C05478=1167.973,405.826,-85.740,-176.090,9.388,148.780
C05479=1167.977,405.579,-85.703,-176.089,9.386,148.779
C05480=1167.980,405.332,-85.667,-176.089,9.384,148.778
C05481=1167.985,405.085,-85.630,-176.088,9.382,148.778
C05482=1167.988,404.838,-85.594,-176.088,9.380,148.777
C05483=1167.992,404.590,-85.558,-176.088,9.378,148.776
C05484=1167.996,404.343,-85.522,-176.087,9.376,148.776
C05485=1168.000,404.095,-85.486,-176.087,9.373,148.775
C05486=1168.003,403.848,-85.449,-176.086,9.372,148.774
C05487=1168.008,403.600,-85.413,-176.086,9.369,148.774
C05488=1168.011,403.354,-85.377,-176.086,9.368,148.773
C05489=1168.016,403.106,-85.341,-176.086,9.365,148.773
C05490=1168.019,402.859,-85.304,-176.085,9.363,148.772
C05491=1168.023,402.611,-85.268,-176.085,9.361,148.771
C05492=1168.027,402.364,-85.231,-176.084,9.359,148.771
C05493=1168.031,402.116,-85.196,-176.084,9.357,148.770
C05494=1168.035,401.869,-85.159,-176.083,9.355,148.769
C05495=1168.039,401.622,-85.124,-176.083,9.352,148.768
C05496=1168.043,401.375,-85.087,-176.082,9.350,148.768
C05497=1168.047,401.127,-85.051,-176.082,9.348,148.767
C05498=1168.051,400.880,-85.014,-176.081,9.346,148.766
C05499=1168.054,400.632,-84.979,-176.081,9.344,148.766
C05500=1168.058,400.385,-84.942,-176.081,9.341,148.765
C05501=1168.062,400.138,-84.906,-176.080,9.339,148.764
C05502=1168.067,399.891,-84.870,-176.080,9.337,148.764
C05503=1168.070,399.644,-84.834,-176.080,9.334,148.763
C05504=1168.075,399.396,-84.797,-176.079,9.332,148.762
C05505=1168.078,399.149,-84.762,-176.079,9.330,148.762
C05506=1168.082,398.902,-84.725,-176.079,9.327,148.761
C05507=1168.086,398.654,-84.689,-176.078,9.326,148.760
C05508=1168.090,398.407,-84.653,-176.078,9.323,148.759
C05509=1168.094,398.160,-84.617,-176.078,9.320,148.759
C05510=1168.098,397.912,-84.580,-176.078,9.317,148.758
C05511=1168.101,397.665,-84.545,-176.077,9.316,148.757
C05512=1168.106,397.417,-84.508,-176.077,9.313,148.757
C05513=1168.109,397.170,-84.472,-176.077,9.311,148.756
C05514=1168.113,396.923,-84.437,-176.076,9.308,148.755
C05515=1168.117,396.676,-84.400,-176.076,9.305,148.754
C05516=1168.121,396.428,-84.364,-176.075,9.304,148.754
C05517=1168.125,396.181,-84.327,-176.075,9.301,148.753
C05518=1168.128,395.933,-84.292,-176.075,9.298,148.752
C05519=1168.133,395.686,-84.255,-176.075,9.296,148.751
C05520=1168.136,395.439,-84.219,-176.074,9.293,148.751
C05521=1168.141,395.191,-84.183,-176.074,9.291,148.750
C05522=1168.144,394.944,-84.147,-176.074,9.288,148.749
C05523=1168.148,394.696,-84.111,-176.074,9.285,148.749
C05524=1168.152,394.449,-84.075,-176.074,9.283,148.748
C05525=1168.156,394.201,-84.038,-176.073,9.280,148.747
C05526=1168.160,393.955,-84.003,-176.073,9.277,148.746
C05527=1168.164,393.708,-83.967,-176.073,9.275,148.746
C05528=1168.168,393.460,-83.931,-176.073,9.272,148.745
C05529=1168.171,393.213,-83.895,-176.073,9.270,148.744
C05530=1168.176,392.965,-83.859,-176.073,9.267,148.743
C05531=1168.180,392.718,-83.823,-176.072,9.265,148.743
C05532=1168.184,392.471,-83.786,-176.073,9.261,148.742
C05533=1168.187,392.223,-83.751,-176.072,9.258,148.741
C05534=1168.191,391.938,-83.708,-176.072,9.256,148.740
C05535=1168.196,391.653,-83.667,-176.072,9.252,148.739
C05536=1168.201,391.368,-83.626,-176.073,9.249,148.739
C05537=1168.205,391.083,-83.584,-176.072,9.246,148.738
C05538=1168.209,390.835,-83.549,-176.072,9.242,148.737
C05539=1168.213,390.588,-83.512,-176.072,9.240,148.736
C05540=1168.216,390.341,-83.476,-176.072,9.237,148.735
C05541=1168.221,390.093,-83.441,-176.073,9.234,148.735
C05542=1168.225,389.847,-83.404,-176.072,9.231,148.734
C05543=1168.228,389.599,-83.369,-176.073,9.228,148.733
C05544=1168.233,389.351,-83.333,-176.073,9.225,148.732
C05545=1168.236,389.104,-83.297,-176.073,9.222,148.731
C05546=1168.241,388.857,-83.260,-176.073,9.219,148.731
C05547=1168.244,388.609,-83.225,-176.073,9.216,148.730
C05548=1168.248,388.362,-83.189,-176.073,9.213,148.729
C05549=1168.252,388.114,-83.152,-176.073,9.210,148.729
C05550=1168.256,387.867,-83.117,-176.073,9.207,148.728
C05551=1168.259,387.619,-83.081,-176.074,9.204,148.727
C05552=1168.264,387.372,-83.045,-176.074,9.201,148.726
C05553=1168.268,387.125,-83.009,-176.075,9.197,148.726
C05554=1168.271,386.878,-82.974,-176.075,9.195,148.725
C05555=1168.276,386.630,-82.937,-176.075,9.191,148.724
C05556=1168.279,386.383,-82.902,-176.075,9.188,148.723
C05557=1168.283,386.136,-82.866,-176.076,9.185,148.723
C05558=1168.287,385.888,-82.829,-176.076,9.181,148.722
C05559=1168.291,385.640,-82.794,-176.077,9.178,148.721
C05560=1168.294,385.393,-82.758,-176.077,9.176,148.721
C05561=1168.299,385.146,-82.723,-176.077,9.172,148.720
C05562=1168.303,384.899,-82.686,-176.078,9.169,148.719
C05563=1168.306,384.651,-82.651,-176.078,9.165,148.718
C05564=1168.311,384.404,-82.615,-176.080,9.161,148.718
C05565=1168.315,384.156,-82.579,-176.080,9.158,148.717
C05566=1168.318,383.909,-82.544,-176.081,9.155,148.716
C05567=1168.322,383.661,-82.508,-176.081,9.152,148.716
C05568=1168.327,383.415,-82.471,-176.082,9.148,148.715
C05569=1168.330,383.167,-82.436,-176.083,9.145,148.714
C05570=1168.334,382.920,-82.400,-176.083,9.142,148.713
C05571=1168.338,382.672,-82.364,-176.084,9.138,148.713
C05572=1168.342,382.424,-82.329,-176.085,9.134,148.712
C05573=1168.346,382.177,-82.293,-176.085,9.131,148.711
C05574=1168.349,381.929,-82.258,-176.086,9.128,148.711
C05575=1168.354,381.682,-82.222,-176.087,9.124,148.710
C05576=1168.358,381.435,-82.186,-176.088,9.121,148.709
C05577=1168.362,381.187,-82.151,-176.089,9.118,148.709
C05578=1168.365,380.940,-82.115,-176.090,9.113,148.708
C05579=1168.370,380.692,-82.079,-176.091,9.110,148.707
C05580=1168.374,380.445,-82.044,-176.092,9.106,148.707
C05581=1168.377,380.198,-82.008,-176.093,9.103,148.706
C05582=1168.381,379.951,-81.972,-176.093,9.100,148.705
C05583=1168.385,379.703,-81.937,-176.095,9.096,148.705
C05584=1168.389,379.455,-81.900,-176.095,9.093,148.704
C05585=1168.394,379.208,-81.866,-176.097,9.089,148.703
C05586=1168.397,378.960,-81.830,-176.098,9.085,148.703
C05587=1168.401,378.713,-81.795,-176.099,9.082,148.702
C05588=1168.405,378.465,-81.759,-176.100,9.078,148.701
C05589=1168.409,378.218,-81.723,-176.101,9.075,148.701
C05590=1168.413,377.971,-81.688,-176.103,9.071,148.700
C05591=1168.417,377.723,-81.652,-176.104,9.067,148.700
C05592=1168.421,377.476,-81.617,-176.104,9.063,148.699
C05593=1168.424,377.228,-81.581,-176.106,9.060,148.698
C05594=1168.428,376.982,-81.546,-176.108,9.056,148.698
C05595=1168.432,376.734,-81.511,-176.109,9.053,148.697
C05596=1168.436,376.487,-81.475,-176.110,9.049,148.697
C05597=1168.441,376.238,-81.440,-176.111,9.045,148.696
C05598=1168.445,375.991,-81.404,-176.113,9.041,148.695
C05599=1168.448,375.744,-81.369,-176.114,9.038,148.695
C05600=1168.452,375.496,-81.333,-176.115,9.034,148.694
C05601=1168.456,375.249,-81.298,-176.117,9.031,148.694
C05602=1168.460,375.002,-81.263,-176.118,9.027,148.693
C05603=1168.464,374.754,-81.228,-176.120,9.023,148.692
C05604=1168.468,374.506,-81.192,-176.121,9.019,148.692
C05605=1168.471,374.259,-81.157,-176.123,9.016,148.691
C05606=1168.476,374.012,-81.121,-176.124,9.012,148.691
C05607=1168.480,373.764,-81.087,-176.125,9.008,148.690
C05608=1168.483,373.516,-81.051,-176.127,9.005,148.690
C05609=1168.487,373.270,-81.016,-176.129,9.001,148.689
C05610=1168.491,373.022,-80.980,-176.130,8.997,148.689
C05611=1168.495,372.774,-80.946,-176.132,8.993,148.688
C05612=1168.499,372.527,-80.910,-176.134,8.990,148.688
C05613=1168.503,372.280,-80.875,-176.135,8.986,148.687
C05614=1168.507,372.032,-80.840,-176.137,8.982,148.687
C05615=1168.511,371.784,-80.804,-176.138,8.978,148.686
C05616=1168.515,371.537,-80.769,-176.140,8.975,148.686
C05617=1168.519,371.289,-80.734,-176.142,8.971,148.685
C05618=1168.523,371.042,-80.699,-176.144,8.967,148.684
C05619=1168.527,370.794,-80.664,-176.145,8.963,148.684
C05620=1168.531,370.547,-80.629,-176.147,8.960,148.684
C05621=1168.535,370.300,-80.594,-176.150,8.955,148.683
C05622=1168.539,370.052,-80.559,-176.151,8.951,148.683
C05623=1168.543,369.804,-80.523,-176.153,8.948,148.682
C05624=1168.547,369.557,-80.489,-176.155,8.944,148.682
C05625=1168.551,369.309,-80.453,-176.157,8.941,148.681
C05626=1168.555,369.061,-80.418,-176.159,8.937,148.681
C05627=1168.559,368.815,-80.383,-176.160,8.933,148.680
C05628=1168.562,368.567,-80.349,-176.162,8.929,148.680
C05629=1168.567,368.320,-80.314,-176.164,8.925,148.679
C05630=1168.571,368.072,-80.279,-176.166,8.922,148.679
C05631=1168.574,367.824,-80.243,-176.168,8.918,148.678
C05632=1168.579,367.577,-80.209,-176.170,8.914,148.678
C05633=1168.583,367.329,-80.173,-176.172,8.910,148.678
C05634=1168.587,367.082,-80.139,-176.174,8.907,148.677
C05635=1168.591,366.834,-80.104,-176.176,8.903,148.677
C05636=1168.594,366.587,-80.069,-176.178,8.899,148.676
C05637=1168.599,366.339,-80.035,-176.180,8.896,148.676
C05638=1168.603,366.057,-79.995,-176.182,8.891,148.676
C05639=1168.607,365.775,-79.955,-176.185,8.887,148.675
C05640=1168.612,365.493,-79.916,-176.187,8.882,148.675
C05641=1168.616,365.211,-79.876,-176.190,8.878,148.674
C05642=1168.620,364.962,-79.841,-176.192,8.874,148.674
C05643=1168.625,364.715,-79.806,-176.194,8.871,148.673
C05644=1168.628,364.468,-79.771,-176.196,8.867,148.673
C05645=1168.632,364.220,-79.737,-176.198,8.863,148.673
C05646=1168.636,363.972,-79.702,-176.200,8.860,148.672
C05647=1168.641,363.725,-79.668,-176.203,8.855,148.672
C05648=1168.644,363.478,-79.633,-176.205,8.852,148.671
C05649=1168.648,363.230,-79.598,-176.207,8.849,148.671
C05650=1168.652,362.982,-79.564,-176.209,8.844,148.671
C05651=1168.656,362.735,-79.530,-176.211,8.840,148.670
C05652=1168.660,362.487,-79.495,-176.214,8.837,148.670
C05653=1168.665,362.239,-79.460,-176.216,8.833,148.670
C05654=1168.668,361.992,-79.425,-176.218,8.829,148.669
C05655=1168.672,361.745,-79.391,-176.220,8.826,148.669
C05656=1168.676,361.497,-79.356,-176.223,8.822,148.669
C05657=1168.680,361.250,-79.322,-176.225,8.818,148.668
C05658=1168.684,361.002,-79.287,-176.227,8.815,148.668
C05659=1168.688,360.754,-79.253,-176.230,8.810,148.668
C05660=1168.692,360.506,-79.219,-176.232,8.807,148.667
C05661=1168.696,360.259,-79.184,-176.234,8.803,148.667
C05662=1168.700,360.011,-79.150,-176.237,8.799,148.667
C05663=1168.704,359.764,-79.116,-176.239,8.796,148.666
C05664=1168.709,359.516,-79.081,-176.241,8.792,148.666
C05665=1168.712,359.268,-79.047,-176.244,8.788,148.666
C05666=1168.716,359.021,-79.012,-176.245,8.785,148.665
C05667=1168.720,358.773,-78.978,-176.248,8.781,148.665
C05668=1168.724,358.526,-78.944,-176.251,8.777,148.665
C05669=1168.727,358.278,-78.909,-176.252,8.774,148.664
C05670=1168.732,358.031,-78.875,-176.255,8.770,148.664
C05671=1168.736,357.783,-78.841,-176.258,8.766,148.664
C05672=1168.740,357.535,-78.806,-176.259,8.763,148.663
C05673=1168.744,357.288,-78.772,-176.262,8.759,148.663
C05674=1168.748,357.039,-78.738,-176.265,8.755,148.663
C05675=1168.752,356.792,-78.704,-176.266,8.752,148.663
C05676=1168.756,356.545,-78.670,-176.269,8.748,148.662
C05677=1168.760,356.297,-78.636,-176.272,8.744,148.662
C05678=1168.764,356.050,-78.601,-176.274,8.741,148.662
C05679=1168.768,355.803,-78.567,-176.276,8.737,148.661
C05680=1168.772,355.554,-78.533,-176.278,8.734,148.661
C05681=1168.776,355.307,-78.499,-176.281,8.730,148.661
C05682=1168.780,355.060,-78.465,-176.283,8.727,148.661
C05683=1168.784,354.812,-78.431,-176.285,8.723,148.660
C05684=1168.788,354.564,-78.398,-176.288,8.719,148.660
C05685=1168.793,354.316,-78.363,-176.290,8.716,148.660
C05686=1168.796,354.069,-78.329,-176.292,8.712,148.660
C05687=1168.801,353.821,-78.295,-176.295,8.708,148.659
C05688=1168.805,353.573,-78.261,-176.297,8.705,148.659
C05689=1168.808,353.326,-78.227,-176.299,8.701,148.659
C05690=1168.813,353.078,-78.193,-176.302,8.698,148.658
C05691=1168.817,352.830,-78.159,-176.305,8.694,148.658
C05692=1168.820,352.583,-78.125,-176.306,8.690,148.658
C05693=1168.825,352.335,-78.091,-176.309,8.687,148.658
C05694=1168.828,352.088,-78.057,-176.312,8.683,148.657
C05695=1168.833,351.840,-78.024,-176.314,8.680,148.657
C05696=1168.837,351.592,-77.989,-176.316,8.676,148.657
C05697=1168.841,351.344,-77.956,-176.318,8.673,148.657
C05698=1168.845,351.097,-77.922,-176.321,8.669,148.656
C05699=1168.849,350.849,-77.889,-176.323,8.665,148.656
C05700=1168.853,350.601,-77.854,-176.325,8.662,148.656
C05701=1168.857,350.353,-77.821,-176.328,8.658,148.656
C05702=1168.861,350.106,-77.787,-176.331,8.655,148.655
C05703=1168.865,349.858,-77.754,-176.333,8.651,148.655
C05704=1168.869,349.610,-77.719,-176.335,8.648,148.655
C05705=1168.873,349.363,-77.686,-176.338,8.643,148.654
C05706=1168.877,349.115,-77.652,-176.340,8.640,148.654
C05707=1168.881,348.868,-77.619,-176.342,8.637,148.654
C05708=1168.886,348.620,-77.586,-176.344,8.634,148.654
C05709=1168.889,348.372,-77.551,-176.347,8.629,148.653
C05710=1168.893,348.124,-77.518,-176.350,8.626,148.653
C05711=1168.897,347.876,-77.485,-176.352,8.623,148.653
C05712=1168.901,347.629,-77.451,-176.354,8.620,148.653
C05713=1168.906,347.381,-77.417,-176.357,8.615,148.653
C05714=1168.910,347.134,-77.384,-176.359,8.612,148.652
C05715=1168.913,346.886,-77.350,-176.362,8.609,148.652
C05716=1168.917,346.638,-77.317,-176.364,8.606,148.652
C05717=1168.922,346.390,-77.284,-176.367,8.601,148.652
C05718=1168.926,346.143,-77.250,-176.369,8.598,148.651
C05719=1168.930,345.895,-77.216,-176.371,8.595,148.651
C05720=1168.934,345.647,-77.183,-176.374,8.592,148.651
C05721=1168.939,345.400,-77.150,-176.376,8.587,148.651
C05722=1168.942,345.151,-77.116,-176.379,8.584,148.651
C05723=1168.946,344.903,-77.083,-176.381,8.581,148.650
C05724=1168.950,344.656,-77.049,-176.383,8.578,148.650
C05725=1168.954,344.409,-77.016,-176.386,8.573,148.650
C05726=1168.958,344.161,-76.983,-176.388,8.570,148.650
C05727=1168.962,343.913,-76.950,-176.391,8.567,148.649
C05728=1168.967,343.665,-76.917,-176.393,8.564,148.649
C05729=1168.971,343.418,-76.883,-176.395,8.560,148.649
C05730=1168.975,343.170,-76.850,-176.398,8.556,148.649
C05731=1168.979,342.922,-76.817,-176.400,8.553,148.649
C05732=1168.983,342.674,-76.784,-176.403,8.550,148.648
C05733=1168.987,342.426,-76.750,-176.405,8.546,148.648
C05734=1168.991,342.178,-76.717,-176.408,8.542,148.648
C05735=1168.995,341.931,-76.684,-176.410,8.539,148.648
C05736=1168.999,341.683,-76.651,-176.412,8.536,148.647
C05737=1169.003,341.435,-76.618,-176.415,8.532,148.647
C05738=1169.007,341.187,-76.585,-176.417,8.529,148.647
C05739=1169.012,340.940,-76.551,-176.420,8.525,148.647
C05740=1169.016,340.692,-76.518,-176.422,8.522,148.647
C05741=1169.020,340.444,-76.485,-176.424,8.518,148.646
C05742=1169.024,340.165,-76.448,-176.428,8.514,148.646
C05743=1169.030,339.886,-76.410,-176.430,8.511,148.646
C05744=1169.034,339.606,-76.373,-176.433,8.507,148.646
C05745=1169.038,339.327,-76.336,-176.436,8.503,148.646
C05746=1169.042,339.079,-76.303,-176.438,8.500,148.645
C05747=1169.046,338.832,-76.270,-176.440,8.496,148.645
C05748=1169.051,338.583,-76.237,-176.443,8.492,148.645
C05749=1169.055,338.335,-76.204,-176.445,8.489,148.645
C05750=1169.059,338.088,-76.171,-176.448,8.486,148.645
C05751=1169.062,337.840,-76.138,-176.450,8.483,148.645
C05752=1169.067,337.593,-76.105,-176.453,8.479,148.644
C05753=1169.071,337.344,-76.073,-176.455,8.476,148.644
C05754=1169.075,337.096,-76.040,-176.458,8.472,148.644
C05755=1169.079,336.849,-76.006,-176.460,8.469,148.644
C05756=1169.083,336.601,-75.974,-176.463,8.466,148.644
C05757=1169.087,336.353,-75.941,-176.465,8.462,148.643
C05758=1169.091,336.105,-75.908,-176.467,8.459,148.643
C05759=1169.095,335.858,-75.875,-176.470,8.455,148.643
C05760=1169.099,335.609,-75.843,-176.473,8.452,148.643
C05761=1169.103,335.362,-75.810,-176.475,8.448,148.643
C05762=1169.108,335.115,-75.777,-176.478,8.445,148.643
C05763=1169.112,334.866,-75.745,-176.480,8.442,148.642
C05764=1169.116,334.619,-75.712,-176.482,8.439,148.642
C05765=1169.120,334.371,-75.680,-176.485,8.435,148.642
C05766=1169.124,334.123,-75.647,-176.487,8.431,148.642
C05767=1169.129,333.875,-75.614,-176.490,8.428,148.642
C05768=1169.132,333.627,-75.582,-176.492,8.425,148.641
C05769=1169.136,333.379,-75.549,-176.495,8.422,148.641
C05770=1169.141,333.131,-75.516,-176.497,8.418,148.641
C05771=1169.144,332.884,-75.484,-176.500,8.415,148.641
C05772=1169.149,332.636,-75.452,-176.503,8.411,148.641
C05773=1169.153,332.388,-75.418,-176.505,8.408,148.641
C05774=1169.157,332.140,-75.387,-176.507,8.405,148.640
C05775=1169.161,331.892,-75.353,-176.510,8.402,148.640
C05776=1169.165,331.644,-75.322,-176.512,8.398,148.640
C05777=1169.169,331.396,-75.289,-176.514,8.395,148.640
C05778=1169.174,331.149,-75.256,-176.517,8.391,148.640
C05779=1169.178,330.901,-75.224,-176.520,8.388,148.640
C05780=1169.182,330.653,-75.191,-176.522,8.385,148.640
C05781=1169.186,330.405,-75.159,-176.525,8.381,148.639
C05782=1169.190,330.157,-75.127,-176.527,8.378,148.639
C05783=1169.194,329.909,-75.094,-176.530,8.375,148.639
C05784=1169.199,329.662,-75.062,-176.532,8.372,148.639
C05785=1169.203,329.413,-75.030,-176.535,8.368,148.639
C05786=1169.206,329.166,-74.997,-176.537,8.365,148.639
C05787=1169.211,328.918,-74.965,-176.540,8.361,148.639
C05788=1169.215,328.670,-74.933,-176.542,8.358,148.638
C05789=1169.219,328.423,-74.900,-176.544,8.355,148.638
C05790=1169.223,328.175,-74.868,-176.547,8.352,148.638
C05791=1169.227,327.926,-74.836,-176.549,8.349,148.638
C05792=1169.231,327.678,-74.804,-176.552,8.344,148.638
C05793=1169.236,327.431,-74.772,-176.555,8.341,148.638
C05794=1169.240,327.183,-74.740,-176.557,8.338,148.637
C05795=1169.244,326.935,-74.707,-176.560,8.335,148.637
C05796=1169.248,326.687,-74.675,-176.562,8.332,148.637
C05797=1169.252,326.439,-74.644,-176.565,8.329,148.637
C05798=1169.257,326.191,-74.611,-176.567,8.325,148.637
C05799=1169.260,325.943,-74.579,-176.570,8.322,148.637
C05800=1169.264,325.695,-74.546,-176.572,8.318,148.637
C05801=1169.269,325.448,-74.515,-176.575,8.315,148.636
C05802=1169.273,325.200,-74.482,-176.577,8.312,148.636
C05803=1169.277,324.952,-74.451,-176.580,8.309,148.636
C05804=1169.281,324.704,-74.419,-176.582,8.305,148.636
C05805=1169.286,324.456,-74.387,-176.585,8.302,148.636
C05806=1169.289,324.208,-74.355,-176.587,8.299,148.636
C05807=1169.293,323.960,-74.323,-176.590,8.296,148.636
C05808=1169.298,323.712,-74.291,-176.592,8.293,148.636
C05809=1169.302,323.464,-74.259,-176.595,8.289,148.635
C05810=1169.305,323.216,-74.227,-176.598,8.286,148.635
C05811=1169.311,322.968,-74.195,-176.600,8.282,148.635
C05812=1169.314,322.720,-74.163,-176.603,8.279,148.635
C05813=1169.318,322.472,-74.131,-176.605,8.276,148.635
C05814=1169.322,322.225,-74.100,-176.607,8.273,148.635
C05815=1169.327,321.977,-74.067,-176.610,8.270,148.635
C05816=1169.330,321.729,-74.036,-176.612,8.267,148.635
C05817=1169.335,321.481,-74.004,-176.615,8.264,148.635
C05818=1169.339,321.233,-73.973,-176.617,8.260,148.634
C05819=1169.343,320.984,-73.941,-176.620,8.257,148.634
C05820=1169.347,320.737,-73.909,-176.623,8.253,148.634
C05821=1169.351,320.489,-73.877,-176.625,8.250,148.634
C05822=1169.355,320.242,-73.846,-176.628,8.247,148.634
C05823=1169.360,319.993,-73.813,-176.630,8.244,148.634
C05824=1169.364,319.745,-73.782,-176.632,8.240,148.634
C05825=1169.368,319.497,-73.751,-176.635,8.237,148.634
C05826=1169.372,319.249,-73.719,-176.637,8.234,148.633
C05827=1169.376,319.002,-73.687,-176.640,8.231,148.633
C05828=1169.381,318.753,-73.656,-176.642,8.228,148.633
C05829=1169.385,318.505,-73.624,-176.645,8.225,148.633
C05830=1169.389,318.258,-73.592,-176.648,8.221,148.633
C05831=1169.393,318.009,-73.561,-176.651,8.218,148.633
C05832=1169.397,317.762,-73.530,-176.653,8.214,148.633
C05833=1169.401,317.513,-73.498,-176.655,8.211,148.633
C05834=1169.405,317.266,-73.466,-176.658,8.208,148.633
C05835=1169.409,317.017,-73.435,-176.660,8.205,148.632
C05836=1169.414,316.770,-73.403,-176.663,8.202,148.633
C05837=1169.418,316.521,-73.372,-176.665,8.198,148.632
C05838=1169.422,316.273,-73.340,-176.668,8.196,148.632
C05839=1169.426,316.026,-73.309,-176.670,8.192,148.632
C05840=1169.430,315.777,-73.278,-176.673,8.189,148.632
C05841=1169.435,315.530,-73.246,-176.675,8.186,148.632
C05842=1169.439,315.281,-73.215,-176.678,8.183,148.632
C05843=1169.443,315.034,-73.184,-176.680,8.180,148.632
C05844=1169.447,314.785,-73.152,-176.683,8.177,148.632
C05845=1169.451,314.538,-73.121,-176.686,8.173,148.632
C05846=1169.456,314.261,-73.086,-176.689,8.170,148.632
C05847=1169.461,313.984,-73.052,-176.691,8.166,148.631
C05848=1169.465,313.706,-73.016,-176.694,8.162,148.631
C05849=1169.470,313.430,-72.981,-176.697,8.158,148.631
C05850=1169.475,313.182,-72.950,-176.700,8.155,148.631
C05851=1169.478,312.934,-72.918,-176.703,8.152,148.631
C05852=1169.483,312.686,-72.888,-176.705,8.149,148.631
C05853=1169.487,312.438,-72.856,-176.708,8.146,148.631
C05854=1169.491,312.190,-72.825,-176.710,8.143,148.631
C05855=1169.496,311.942,-72.794,-176.713,8.140,148.631
C05856=1169.500,311.694,-72.762,-176.715,8.137,148.631
C05857=1169.503,311.446,-72.732,-176.718,8.134,148.631
C05858=1169.507,311.197,-72.701,-176.720,8.130,148.630
C05859=1169.512,310.950,-72.670,-176.723,8.127,148.630
C05860=1169.516,310.701,-72.638,-176.725,8.124,148.630
C05861=1169.520,310.453,-72.608,-176.728,8.121,148.630
C05862=1169.525,310.205,-72.577,-176.730,8.118,148.630
C05863=1169.529,309.957,-72.545,-176.733,8.115,148.630
C05864=1169.533,309.709,-72.514,-176.736,8.112,148.630
C05865=1169.538,309.461,-72.484,-176.738,8.108,148.630
C05866=1169.541,309.213,-72.453,-176.741,8.106,148.630
C05867=1169.546,308.966,-72.421,-176.743,8.102,148.630
C05868=1169.550,308.717,-72.390,-176.746,8.099,148.630
C05869=1169.554,308.469,-72.360,-176.748,8.096,148.630
C05870=1169.559,308.221,-72.329,-176.751,8.093,148.630
C05871=1169.562,307.973,-72.298,-176.753,8.090,148.629
C05872=1169.567,307.725,-72.268,-176.756,8.087,148.629
C05873=1169.571,307.477,-72.236,-176.758,8.084,148.629
C05874=1169.575,307.229,-72.205,-176.761,8.080,148.629
C05875=1169.580,306.981,-72.174,-176.763,8.077,148.629
C05876=1169.583,306.733,-72.144,-176.766,8.074,148.629
C05877=1169.587,306.485,-72.113,-176.769,8.070,148.629
C05878=1169.592,306.237,-72.082,-176.772,8.067,148.629
C05879=1169.597,305.989,-72.051,-176.774,8.064,148.629
C05880=1169.600,305.740,-72.021,-176.777,8.061,148.629
C05881=1169.605,305.492,-71.990,-176.779,8.058,148.629
C05882=1169.609,305.244,-71.959,-176.782,8.055,148.629
C05883=1169.614,304.996,-71.929,-176.785,8.052,148.629
C05884=1169.617,304.748,-71.898,-176.787,8.049,148.629
C05885=1169.622,304.500,-71.867,-176.790,8.046,148.629
C05886=1169.626,304.252,-71.836,-176.792,8.042,148.628
C05887=1169.630,304.004,-71.806,-176.795,8.039,148.628
C05888=1169.634,303.756,-71.775,-176.797,8.036,148.628
C05889=1169.639,303.508,-71.744,-176.800,8.033,148.628
C05890=1169.643,303.260,-71.714,-176.802,8.030,148.628
C05891=1169.647,303.011,-71.684,-176.805,8.027,148.628
C05892=1169.652,302.763,-71.653,-176.807,8.024,148.628
C05893=1169.656,302.515,-71.623,-176.810,8.021,148.628
C05894=1169.660,302.267,-71.592,-176.812,8.017,148.628
C05895=1169.664,302.020,-71.562,-176.815,8.015,148.628
C05896=1169.668,301.771,-71.531,-176.818,8.012,148.628
C05897=1169.673,301.523,-71.501,-176.820,8.008,148.628
C05898=1169.677,301.275,-71.471,-176.823,8.005,148.628
C05899=1169.681,301.027,-71.440,-176.826,8.002,148.628
C05900=1169.685,300.779,-71.409,-176.828,7.999,148.628
C05901=1169.690,300.530,-71.379,-176.831,7.996,148.628
C05902=1169.693,300.282,-71.349,-176.833,7.993,148.628
C05903=1169.698,300.034,-71.318,-176.836,7.990,148.628
C05904=1169.702,299.787,-71.288,-176.838,7.988,148.628
C05905=1169.707,299.538,-71.258,-176.841,7.985,148.628
C05906=1169.710,299.290,-71.228,-176.843,7.981,148.628
C05907=1169.715,299.042,-71.197,-176.846,7.978,148.628
C05908=1169.719,298.794,-71.167,-176.848,7.975,148.628
C05909=1169.724,298.546,-71.137,-176.851,7.972,148.627
C05910=1169.727,298.298,-71.106,-176.853,7.969,148.627
C05911=1169.732,298.049,-71.076,-176.856,7.966,148.627
C05912=1169.736,297.801,-71.046,-176.858,7.963,148.627
C05913=1169.741,297.552,-71.016,-176.861,7.960,148.627
C05914=1169.744,297.305,-70.986,-176.864,7.957,148.627
C05915=1169.749,297.057,-70.956,-176.867,7.954,148.627
C05916=1169.753,296.809,-70.925,-176.869,7.951,148.627
C05917=1169.757,296.561,-70.895,-176.872,7.948,148.627
C05918=1169.762,296.312,-70.865,-176.874,7.945,148.627
C05919=1169.766,296.065,-70.835,-176.877,7.941,148.627
C05920=1169.769,295.816,-70.805,-176.879,7.938,148.627
C05921=1169.774,295.568,-70.774,-176.882,7.935,148.627
C05922=1169.778,295.320,-70.745,-176.884,7.932,148.627
C05923=1169.782,295.072,-70.715,-176.887,7.929,148.627
C05924=1169.787,294.823,-70.685,-176.890,7.926,148.627
C05925=1169.791,294.575,-70.655,-176.893,7.923,148.627
C05926=1169.795,294.327,-70.625,-176.895,7.920,148.627
C05927=1169.800,294.079,-70.595,-176.898,7.917,148.627
C05928=1169.804,293.831,-70.565,-176.900,7.914,148.627
C05929=1169.808,293.583,-70.535,-176.903,7.911,148.627
C05930=1169.813,293.334,-70.505,-176.906,7.908,148.627
C05931=1169.817,293.087,-70.475,-176.908,7.905,148.627
C05932=1169.821,292.838,-70.446,-176.910,7.903,148.627
C05933=1169.826,292.590,-70.416,-176.913,7.900,148.627
C05934=1169.830,292.342,-70.386,-176.915,7.896,148.627
C05935=1169.834,292.094,-70.356,-176.918,7.893,148.627
C05936=1169.838,291.846,-70.327,-176.921,7.890,148.627
C05937=1169.842,291.597,-70.297,-176.924,7.887,148.627
C05938=1169.846,291.349,-70.266,-176.926,7.884,148.627
C05939=1169.851,291.100,-70.237,-176.929,7.881,148.627
C05940=1169.855,290.852,-70.207,-176.931,7.878,148.627
C05941=1169.859,290.604,-70.178,-176.934,7.875,148.627
C05942=1169.864,290.356,-70.147,-176.936,7.872,148.627
C05943=1169.868,290.108,-70.118,-176.939,7.869,148.627
C05944=1169.873,289.860,-70.088,-176.942,7.866,148.627
C05945=1169.877,289.612,-70.059,-176.945,7.863,148.627
C05946=1169.881,289.364,-70.030,-176.947,7.860,148.626
C05947=1169.885,289.115,-70.000,-176.949,7.858,148.627
C05948=1169.889,288.868,-69.970,-176.952,7.855,148.627
C05949=1169.894,288.619,-69.940,-176.955,7.852,148.627
C05950=1169.898,288.344,-69.908,-176.958,7.848,148.627
C05951=1169.903,288.069,-69.875,-176.961,7.845,148.627
C05952=1169.908,287.794,-69.842,-176.963,7.842,148.626
C05953=1169.913,287.520,-69.809,-176.966,7.838,148.626
C05954=1169.917,287.272,-69.780,-176.969,7.835,148.626
C05955=1169.921,287.023,-69.750,-176.972,7.832,148.627
C05956=1169.925,286.775,-69.721,-176.974,7.830,148.627
C05957=1169.930,286.527,-69.691,-176.976,7.826,148.626
C05958=1169.934,286.278,-69.662,-176.979,7.823,148.626
C05959=1169.938,286.030,-69.632,-176.982,7.820,148.626
C05960=1169.942,285.782,-69.603,-176.984,7.817,148.627
C05961=1169.947,285.533,-69.574,-176.987,7.814,148.627
C05962=1169.951,285.285,-69.545,-176.990,7.811,148.627
C05963=1169.956,285.037,-69.516,-176.992,7.808,148.626
C05964=1169.960,284.789,-69.486,-176.995,7.805,148.626
C05965=1169.964,284.541,-69.457,-176.998,7.802,148.627
C05966=1169.968,284.292,-69.427,-177.000,7.800,148.627
C05967=1169.972,284.044,-69.398,-177.003,7.797,148.627
C05968=1169.977,283.796,-69.368,-177.005,7.794,148.627
C05969=1169.981,283.548,-69.339,-177.008,7.791,148.626
C05970=1169.986,283.299,-69.310,-177.010,7.788,148.627
C05971=1169.990,283.051,-69.281,-177.013,7.785,148.627
C05972=1169.994,282.803,-69.252,-177.016,7.782,148.627
C05973=1169.998,282.555,-69.222,-177.019,7.779,148.627
C05974=1170.003,282.306,-69.193,-177.021,7.776,148.627
C05975=1170.008,282.058,-69.164,-177.024,7.773,148.627
C05976=1170.012,281.810,-69.135,-177.026,7.771,148.627
C05977=1170.016,281.562,-69.105,-177.029,7.768,148.627
C05978=1170.020,281.313,-69.077,-177.031,7.765,148.627
C05979=1170.024,281.065,-69.048,-177.034,7.762,148.627
C05980=1170.029,280.817,-69.019,-177.037,7.759,148.627
C05981=1170.033,280.569,-68.989,-177.040,7.756,148.627
C05982=1170.037,280.320,-68.960,-177.042,7.752,148.627
C05983=1170.042,280.072,-68.931,-177.045,7.749,148.627
C05984=1170.046,279.823,-68.902,-177.047,7.747,148.627
C05985=1170.050,279.576,-68.874,-177.050,7.744,148.627
C05986=1170.054,279.327,-68.844,-177.052,7.741,148.627
C05987=1170.059,279.079,-68.816,-177.055,7.738,148.627
C05988=1170.063,278.830,-68.786,-177.058,7.735,148.627
C05989=1170.068,278.582,-68.758,-177.060,7.732,148.627
C05990=1170.071,278.334,-68.729,-177.063,7.729,148.627
C05991=1170.076,278.086,-68.699,-177.066,7.726,148.627
C05992=1170.080,277.837,-68.671,-177.068,7.724,148.627
C05993=1170.085,277.589,-68.642,-177.070,7.721,148.627
C05994=1170.089,277.341,-68.613,-177.073,7.718,148.627
C05995=1170.093,277.093,-68.584,-177.076,7.715,148.627
C05996=1170.098,276.844,-68.556,-177.079,7.712,148.627
C05997=1170.101,276.596,-68.527,-177.081,7.709,148.627
C05998=1170.106,276.348,-68.498,-177.084,7.706,148.627
C05999=1170.110,276.099,-68.469,-177.086,7.704,148.627
C06000=1170.115,275.851,-68.440,-177.089,7.701,148.627
C06001=1170.119,275.602,-68.412,-177.092,7.698,148.627
C06002=1170.123,275.354,-68.383,-177.094,7.695,148.627
C06003=1170.128,275.106,-68.354,-177.097,7.692,148.627
C06004=1170.132,274.858,-68.325,-177.100,7.689,148.627
C06005=1170.136,274.609,-68.297,-177.102,7.687,148.627
C06006=1170.141,274.361,-68.268,-177.105,7.684,148.627
C06007=1170.145,274.113,-68.239,-177.107,7.681,148.627
C06008=1170.149,273.864,-68.211,-177.110,7.678,148.627
C06009=1170.153,273.616,-68.183,-177.113,7.675,148.628
C06010=1170.158,273.368,-68.153,-177.116,7.672,148.628
C06011=1170.163,273.120,-68.125,-177.118,7.670,148.628
C06012=1170.167,272.871,-68.097,-177.120,7.667,148.628
C06013=1170.171,272.622,-68.068,-177.123,7.664,148.628
C06014=1170.175,272.375,-68.040,-177.126,7.661,148.628
C06015=1170.180,272.126,-68.011,-177.129,7.658,148.628
C06016=1170.184,271.877,-67.982,-177.131,7.655,148.628
C06017=1170.188,271.629,-67.954,-177.134,7.653,148.628
C06018=1170.193,271.381,-67.926,-177.136,7.650,148.628
C06019=1170.197,271.133,-67.897,-177.139,7.647,148.628
C06020=1170.201,270.884,-67.869,-177.142,7.644,148.628
C06021=1170.206,270.637,-67.841,-177.145,7.641,148.628
C06022=1170.210,270.388,-67.812,-177.147,7.638,148.628
C06023=1170.214,270.139,-67.784,-177.149,7.635,148.628
C06024=1170.219,269.891,-67.755,-177.152,7.633,148.628
C06025=1170.223,269.642,-67.727,-177.155,7.630,148.628
C06026=1170.228,269.395,-67.698,-177.157,7.627,148.628
C06027=1170.231,269.146,-67.670,-177.160,7.624,148.628
C06028=1170.236,268.898,-67.642,-177.162,7.621,148.628
C06029=1170.240,268.649,-67.614,-177.165,7.618,148.628
C06030=1170.245,268.401,-67.585,-177.168,7.616,148.628
C06031=1170.249,268.153,-67.557,-177.170,7.613,148.629
C06032=1170.253,267.905,-67.529,-177.173,7.610,148.629
C06033=1170.258,267.656,-67.501,-177.175,7.607,148.629
C06034=1170.262,267.408,-67.473,-177.178,7.604,148.629
C06035=1170.267,267.159,-67.444,-177.181,7.602,148.629
C06036=1170.271,266.911,-67.416,-177.184,7.599,148.629
C06037=1170.275,266.663,-67.388,-177.186,7.596,148.629
C06038=1170.280,266.415,-67.360,-177.189,7.593,148.629
C06039=1170.284,266.166,-67.332,-177.191,7.590,148.629
C06040=1170.289,265.917,-67.304,-177.194,7.588,148.629
C06041=1170.293,265.669,-67.276,-177.197,7.585,148.629
C06042=1170.297,265.421,-67.248,-177.200,7.582,148.629
C06043=1170.302,265.172,-67.219,-177.202,7.580,148.629
C06044=1170.306,264.924,-67.192,-177.205,7.577,148.630
C06045=1170.310,264.675,-67.163,-177.208,7.574,148.630
C06046=1170.315,264.427,-67.135,-177.210,7.571,148.630
C06047=1170.319,264.178,-67.108,-177.213,7.569,148.630
C06048=1170.323,263.930,-67.080,-177.215,7.566,148.630
C06049=1170.328,263.682,-67.052,-177.218,7.563,148.630
C06050=1170.332,263.433,-67.023,-177.221,7.560,148.630
C06051=1170.336,263.185,-66.996,-177.224,7.557,148.630
C06052=1170.340,262.936,-66.968,-177.226,7.555,148.630
C06053=1170.346,262.688,-66.940,-177.229,7.552,148.630
C06054=1170.350,262.415,-66.909,-177.231,7.549,148.630
C06055=1170.355,262.141,-66.878,-177.234,7.546,148.630
C06056=1170.360,261.869,-66.848,-177.238,7.542,148.630
C06057=1170.364,261.596,-66.818,-177.241,7.539,148.630
C06058=1170.369,261.348,-66.790,-177.243,7.537,148.631
C06059=1170.373,261.099,-66.761,-177.246,7.534,148.631
C06060=1170.378,260.850,-66.734,-177.248,7.531,148.631
C06061=1170.382,260.603,-66.707,-177.251,7.528,148.631
C06062=1170.386,260.354,-66.678,-177.253,7.526,148.631
C06063=1170.391,260.105,-66.651,-177.256,7.523,148.631
C06064=1170.395,259.857,-66.623,-177.259,7.520,148.631
C06065=1170.399,259.608,-66.596,-177.261,7.517,148.631
C06066=1170.404,259.360,-66.568,-177.264,7.515,148.631
C06067=1170.408,259.111,-66.540,-177.267,7.513,148.631
C06068=1170.412,258.863,-66.513,-177.270,7.510,148.631
C06069=1170.417,258.615,-66.485,-177.272,7.507,148.631
C06070=1170.421,258.366,-66.457,-177.275,7.505,148.632
C06071=1170.426,258.118,-66.429,-177.277,7.502,148.632
C06072=1170.430,257.869,-66.402,-177.280,7.499,148.632
C06073=1170.435,257.622,-66.374,-177.283,7.496,148.632
C06074=1170.439,257.372,-66.347,-177.285,7.493,148.632
C06075=1170.443,257.124,-66.320,-177.288,7.491,148.632
C06076=1170.448,256.876,-66.292,-177.291,7.488,148.632
C06077=1170.452,256.627,-66.265,-177.294,7.485,148.632
C06078=1170.456,256.379,-66.237,-177.296,7.483,148.632
C06079=1170.461,256.130,-66.210,-177.299,7.480,148.632
C06080=1170.465,255.882,-66.183,-177.301,7.477,148.632
C06081=1170.469,255.633,-66.154,-177.304,7.474,148.632
C06082=1170.474,255.385,-66.127,-177.306,7.472,148.633
C06083=1170.478,255.137,-66.100,-177.310,7.469,148.633
C06084=1170.483,254.888,-66.073,-177.312,7.466,148.633
C06085=1170.487,254.639,-66.045,-177.314,7.464,148.633
C06086=1170.491,254.391,-66.017,-177.317,7.461,148.633
C06087=1170.496,254.143,-65.990,-177.320,7.458,148.633
C06088=1170.501,253.894,-65.963,-177.323,7.455,148.633
C06089=1170.505,253.645,-65.936,-177.325,7.453,148.633
C06090=1170.509,253.397,-65.908,-177.328,7.450,148.634
C06091=1170.514,253.149,-65.881,-177.331,7.447,148.634
C06092=1170.518,252.900,-65.854,-177.333,7.445,148.634
C06093=1170.522,252.651,-65.826,-177.336,7.442,148.634
C06094=1170.526,252.404,-65.799,-177.339,7.439,148.634
C06095=1170.531,252.155,-65.772,-177.341,7.437,148.634
C06096=1170.535,251.907,-65.745,-177.344,7.435,148.634
C06097=1170.540,251.658,-65.718,-177.347,7.432,148.634
C06098=1170.545,251.410,-65.691,-177.349,7.429,148.634
C06099=1170.549,251.160,-65.664,-177.352,7.426,148.634
C06100=1170.553,250.913,-65.636,-177.354,7.424,148.634
C06101=1170.558,250.664,-65.609,-177.358,7.421,148.635
C06102=1170.562,250.416,-65.582,-177.360,7.419,148.635
C06103=1170.566,250.167,-65.555,-177.363,7.416,148.635
C06104=1170.571,249.919,-65.528,-177.365,7.413,148.635
C06105=1170.575,249.670,-65.501,-177.367,7.411,148.635
C06106=1170.580,249.421,-65.474,-177.371,7.408,148.635
C06107=1170.584,249.173,-65.447,-177.373,7.405,148.635
C06108=1170.588,248.925,-65.420,-177.376,7.403,148.636
C06109=1170.593,248.676,-65.393,-177.378,7.400,148.636
C06110=1170.598,248.428,-65.366,-177.381,7.397,148.636
C06111=1170.602,248.179,-65.339,-177.384,7.395,148.636
C06112=1170.606,247.931,-65.313,-177.387,7.392,148.636
C06113=1170.610,247.682,-65.285,-177.389,7.389,148.636
C06114=1170.615,247.433,-65.258,-177.391,7.387,148.636
C06115=1170.619,247.185,-65.232,-177.394,7.384,148.636
C06116=1170.623,246.936,-65.205,-177.397,7.382,148.637
C06117=1170.628,246.688,-65.177,-177.400,7.379,148.637
C06118=1170.633,246.439,-65.150,-177.402,7.377,148.637
C06119=1170.637,246.191,-65.124,-177.405,7.374,148.637
C06120=1170.641,245.943,-65.097,-177.408,7.372,148.637
C06121=1170.646,245.694,-65.071,-177.411,7.369,148.637
C06122=1170.650,245.445,-65.044,-177.413,7.366,148.637
C06123=1170.655,245.197,-65.017,-177.415,7.364,148.637
C06124=1170.659,244.949,-64.990,-177.419,7.361,148.638
C06125=1170.663,244.700,-64.963,-177.421,7.358,148.638
C06126=1170.668,244.452,-64.936,-177.424,7.356,148.638
C06127=1170.673,244.203,-64.910,-177.426,7.353,148.638
C06128=1170.677,243.955,-64.884,-177.430,7.350,148.638
C06129=1170.682,243.706,-64.857,-177.432,7.348,148.638
C06130=1170.686,243.458,-64.830,-177.435,7.345,148.638
C06131=1170.690,243.208,-64.803,-177.438,7.343,148.639
C06132=1170.695,242.960,-64.776,-177.440,7.341,148.639
C06133=1170.698,242.711,-64.750,-177.443,7.338,148.639
C06134=1170.703,242.463,-64.723,-177.445,7.335,148.639
C06135=1170.708,242.215,-64.697,-177.448,7.333,148.639
C06136=1170.713,241.966,-64.670,-177.451,7.330,148.639
C06137=1170.717,241.718,-64.644,-177.453,7.328,148.639
C06138=1170.721,241.469,-64.618,-177.456,7.325,148.639
C06139=1170.725,241.221,-64.591,-177.459,7.322,148.640
C06140=1170.730,240.972,-64.565,-177.461,7.320,148.640
C06141=1170.734,240.723,-64.538,-177.464,7.317,148.640
C06142=1170.739,240.475,-64.511,-177.467,7.315,148.640
C06143=1170.743,240.226,-64.485,-177.469,7.312,148.640
C06144=1170.748,239.978,-64.458,-177.472,7.309,148.640
C06145=1170.752,239.729,-64.433,-177.475,7.308,148.641
C06146=1170.757,239.480,-64.406,-177.478,7.305,148.641
C06147=1170.761,239.232,-64.380,-177.480,7.302,148.641
C06148=1170.766,238.983,-64.353,-177.483,7.300,148.641
C06149=1170.770,238.735,-64.326,-177.486,7.297,148.641
C06150=1170.774,238.486,-64.300,-177.488,7.295,148.641
C06151=1170.779,238.237,-64.274,-177.491,7.292,148.642
C06152=1170.783,237.988,-64.247,-177.493,7.290,148.642
C06153=1170.788,237.740,-64.222,-177.496,7.287,148.642
C06154=1170.792,237.492,-64.195,-177.499,7.284,148.642
C06155=1170.797,237.243,-64.169,-177.501,7.282,148.642
C06156=1170.801,236.995,-64.142,-177.504,7.279,148.642
C06157=1170.806,236.746,-64.116,-177.507,7.277,148.643
C06158=1170.810,236.474,-64.087,-177.510,7.275,148.643
C06159=1170.815,236.203,-64.059,-177.512,7.272,148.643
C06160=1170.820,235.931,-64.030,-177.516,7.269,148.643
C06161=1170.825,235.659,-64.002,-177.518,7.266,148.643
C06162=1170.829,235.412,-63.976,-177.522,7.263,148.643
C06163=1170.834,235.162,-63.949,-177.524,7.261,148.643
C06164=1170.839,234.914,-63.924,-177.527,7.259,148.644
C06165=1170.842,234.665,-63.897,-177.529,7.256,148.644
C06166=1170.847,234.416,-63.871,-177.532,7.254,148.644
C06167=1170.852,234.168,-63.845,-177.535,7.251,148.644
C06168=1170.856,233.919,-63.820,-177.537,7.249,148.644
C06169=1170.861,233.671,-63.793,-177.540,7.246,148.644
C06170=1170.865,233.422,-63.767,-177.543,7.244,148.645
C06171=1170.870,233.173,-63.741,-177.546,7.241,148.645
C06172=1170.874,232.925,-63.715,-177.548,7.239,148.645
C06173=1170.879,232.677,-63.689,-177.551,7.236,148.645
C06174=1170.883,232.428,-63.663,-177.554,7.233,148.645
C06175=1170.888,232.179,-63.637,-177.556,7.232,148.646
C06176=1170.892,231.930,-63.611,-177.559,7.229,148.646
C06177=1170.897,231.681,-63.585,-177.561,7.226,148.646
C06178=1170.902,231.433,-63.560,-177.565,7.224,148.646
C06179=1170.905,231.185,-63.533,-177.567,7.222,148.646
C06180=1170.910,230.936,-63.508,-177.570,7.219,148.647
C06181=1170.914,230.687,-63.482,-177.572,7.217,148.647
C06182=1170.919,230.439,-63.456,-177.575,7.214,148.647
C06183=1170.924,230.190,-63.430,-177.578,7.212,148.647
C06184=1170.928,229.941,-63.404,-177.580,7.209,148.647
C06185=1170.932,229.693,-63.379,-177.584,7.207,148.647
C06186=1170.937,229.444,-63.353,-177.586,7.205,148.648
C06187=1170.941,229.196,-63.327,-177.589,7.202,148.648
C06188=1170.945,228.947,-63.302,-177.591,7.200,148.648
C06189=1170.950,228.699,-63.276,-177.594,7.197,148.648
C06190=1170.955,228.450,-63.250,-177.597,7.195,148.648
C06191=1170.959,228.201,-63.224,-177.599,7.192,148.648
C06192=1170.964,227.952,-63.198,-177.602,7.190,148.649
C06193=1170.968,227.704,-63.173,-177.605,7.187,148.649
C06194=1170.973,227.455,-63.147,-177.607,7.186,148.649
C06195=1170.977,227.206,-63.122,-177.610,7.183,148.649
C06196=1170.982,226.958,-63.096,-177.612,7.180,148.649
C06197=1170.986,226.709,-63.070,-177.616,7.178,148.650
C06198=1170.990,226.461,-63.045,-177.618,7.176,148.650
C06199=1170.995,226.212,-63.019,-177.621,7.173,148.650
C06200=1171.000,225.963,-62.994,-177.623,7.171,148.650
C06201=1171.004,225.714,-62.969,-177.626,7.168,148.650
C06202=1171.009,225.466,-62.943,-177.629,7.166,148.651
C06203=1171.013,225.217,-62.917,-177.632,7.164,148.651
C06204=1171.017,224.968,-62.892,-177.634,7.161,148.651
C06205=1171.022,224.720,-62.866,-177.637,7.159,148.651
C06206=1171.026,224.471,-62.841,-177.639,7.157,148.651
C06207=1171.031,224.223,-62.816,-177.642,7.154,148.651
C06208=1171.035,223.974,-62.790,-177.645,7.152,148.652
C06209=1171.040,223.725,-62.764,-177.648,7.149,148.652
C06210=1171.045,223.477,-62.739,-177.650,7.147,148.652
C06211=1171.049,223.228,-62.714,-177.653,7.144,148.652
C06212=1171.054,222.980,-62.689,-177.656,7.142,148.653
C06213=1171.058,222.731,-62.663,-177.659,7.140,148.653
C06214=1171.063,222.481,-62.638,-177.661,7.138,148.653
C06215=1171.067,222.233,-62.612,-177.664,7.135,148.653
C06216=1171.072,221.984,-62.587,-177.667,7.133,148.653
C06217=1171.076,221.736,-62.563,-177.669,7.130,148.654
C06218=1171.080,221.487,-62.537,-177.672,7.128,148.654
C06219=1171.085,221.238,-62.511,-177.675,7.125,148.654
C06220=1171.090,220.990,-62.486,-177.677,7.124,148.654
C06221=1171.094,220.741,-62.461,-177.680,7.121,148.654
C06222=1171.099,220.493,-62.435,-177.683,7.119,148.655
C06223=1171.103,220.243,-62.410,-177.686,7.116,148.655
C06224=1171.107,219.996,-62.385,-177.688,7.114,148.655
C06225=1171.112,219.746,-62.360,-177.691,7.111,148.655
C06226=1171.117,219.498,-62.335,-177.694,7.109,148.656
C06227=1171.121,219.249,-62.310,-177.696,7.107,148.656
C06228=1171.126,219.001,-62.285,-177.699,7.105,148.656
C06229=1171.130,218.751,-62.260,-177.701,7.102,148.656
C06230=1171.135,218.503,-62.235,-177.705,7.100,148.656
C06231=1171.139,218.254,-62.210,-177.707,7.098,148.657
C06232=1171.144,218.006,-62.184,-177.710,7.095,148.657
C06233=1171.148,217.757,-62.160,-177.713,7.093,148.657
C06234=1171.153,217.509,-62.134,-177.715,7.090,148.657
C06235=1171.157,217.259,-62.109,-177.718,7.089,148.658
C06236=1171.162,217.011,-62.084,-177.721,7.086,148.658
C06237=1171.166,216.762,-62.060,-177.724,7.084,148.658
C06238=1171.171,216.514,-62.034,-177.726,7.082,148.658
C06239=1171.175,216.264,-62.009,-177.729,7.079,148.658
C06240=1171.180,216.016,-61.985,-177.731,7.077,148.659
C06241=1171.184,215.767,-61.959,-177.734,7.074,148.659
C06242=1171.189,215.518,-61.935,-177.737,7.072,148.659
C06243=1171.193,215.269,-61.910,-177.740,7.070,148.659
C06244=1171.197,215.021,-61.885,-177.742,7.068,148.660
C06245=1171.203,214.773,-61.860,-177.745,7.066,148.660
C06246=1171.206,214.523,-61.836,-177.748,7.063,148.660
C06247=1171.211,214.275,-61.810,-177.750,7.061,148.660
C06248=1171.216,214.026,-61.785,-177.753,7.058,148.661
C06249=1171.220,213.777,-61.761,-177.756,7.056,148.661
C06250=1171.224,213.529,-61.736,-177.759,7.054,148.661
C06251=1171.230,213.280,-61.711,-177.761,7.051,148.661
C06252=1171.234,213.032,-61.687,-177.764,7.050,148.661
C06253=1171.238,212.782,-61.662,-177.767,7.047,148.662
C06254=1171.243,212.534,-61.638,-177.769,7.045,148.662
C06255=1171.247,212.285,-61.612,-177.772,7.042,148.662
C06256=1171.252,212.036,-61.587,-177.774,7.040,148.662
C06257=1171.257,211.788,-61.563,-177.777,7.038,148.663
C06258=1171.261,211.538,-61.538,-177.780,7.035,148.663
C06259=1171.266,211.290,-61.514,-177.783,7.034,148.663
C06260=1171.271,211.041,-61.489,-177.786,7.031,148.663
C06261=1171.274,210.793,-61.464,-177.788,7.029,148.663
C06262=1171.280,210.522,-61.438,-177.791,7.026,148.664
C06263=1171.285,210.252,-61.412,-177.794,7.025,148.664
C06264=1171.289,209.981,-61.384,-177.797,7.022,148.664
C06265=1171.294,209.711,-61.358,-177.800,7.019,148.665
C06266=1171.300,209.462,-61.333,-177.803,7.017,148.665
C06267=1171.303,209.213,-61.309,-177.805,7.014,148.665
C06268=1171.309,208.964,-61.284,-177.808,7.013,148.665
C06269=1171.313,208.716,-61.260,-177.811,7.011,148.666
C06270=1171.317,208.466,-61.235,-177.813,7.008,148.666
C06271=1171.322,208.218,-61.211,-177.816,7.006,148.666
C06272=1171.326,207.969,-61.187,-177.818,7.004,148.666
C06273=1171.331,207.720,-61.162,-177.822,7.001,148.667
C06274=1171.335,207.472,-61.138,-177.824,6.999,148.667
C06275=1171.340,207.223,-61.113,-177.827,6.997,148.667
C06276=1171.345,206.975,-61.089,-177.830,6.995,148.667
C06277=1171.349,206.725,-61.064,-177.832,6.993,148.667
C06278=1171.354,206.477,-61.040,-177.835,6.990,148.668
C06279=1171.358,206.228,-61.016,-177.838,6.988,148.668
C06280=1171.363,205.980,-60.991,-177.840,6.986,148.668
C06281=1171.367,205.730,-60.967,-177.843,6.984,148.669
C06282=1171.371,205.482,-60.942,-177.846,6.982,148.669
C06283=1171.377,205.233,-60.919,-177.848,6.980,148.669
C06284=1171.381,204.984,-60.894,-177.851,6.977,148.669
C06285=1171.386,204.735,-60.869,-177.854,6.975,148.669
C06286=1171.390,204.486,-60.845,-177.857,6.972,148.670
C06287=1171.394,204.238,-60.821,-177.859,6.970,148.670
C06288=1171.399,203.989,-60.798,-177.862,6.968,148.670
C06289=1171.404,203.740,-60.773,-177.865,6.966,148.671
C06290=1171.408,203.491,-60.749,-177.868,6.964,148.671
C06291=1171.412,203.243,-60.725,-177.870,6.962,148.671
C06292=1171.418,202.994,-60.700,-177.873,6.959,148.671
C06293=1171.422,202.745,-60.677,-177.876,6.957,148.672
C06294=1171.427,202.497,-60.653,-177.878,6.955,148.672
C06295=1171.431,202.247,-60.628,-177.881,6.953,148.672
C06296=1171.436,201.998,-60.604,-177.884,6.951,148.672
C06297=1171.440,201.750,-60.580,-177.886,6.949,148.673
C06298=1171.445,201.501,-60.556,-177.889,6.946,148.673
C06299=1171.449,201.253,-60.532,-177.892,6.944,148.673
C06300=1171.455,201.004,-60.508,-177.894,6.942,148.673
C06301=1171.458,200.754,-60.484,-177.897,6.940,148.674
C06302=1171.463,200.505,-60.460,-177.900,6.938,148.674
C06303=1171.467,200.257,-60.436,-177.902,6.936,148.674
C06304=1171.472,200.009,-60.412,-177.905,6.933,148.675
C06305=1171.477,199.759,-60.388,-177.908,6.931,148.675
C06306=1171.482,199.511,-60.364,-177.910,6.929,148.675
C06307=1171.486,199.262,-60.341,-177.914,6.927,148.675
C06308=1171.490,199.013,-60.316,-177.916,6.925,148.676
C06309=1171.495,198.764,-60.292,-177.918,6.923,148.676
C06310=1171.499,198.515,-60.269,-177.921,6.921,148.676
C06311=1171.504,198.267,-60.245,-177.924,6.918,148.676
C06312=1171.509,198.017,-60.221,-177.926,6.916,148.677
C06313=1171.513,197.769,-60.197,-177.929,6.915,148.677
C06314=1171.518,197.520,-60.173,-177.932,6.912,148.677
C06315=1171.523,197.272,-60.149,-177.935,6.910,148.678
C06316=1171.527,197.023,-60.126,-177.937,6.908,148.678
C06317=1171.532,196.774,-60.102,-177.941,6.905,148.678
C06318=1171.536,196.525,-60.079,-177.943,6.904,148.678
C06319=1171.540,196.275,-60.055,-177.945,6.902,148.679
C06320=1171.545,196.027,-60.031,-177.948,6.900,148.679
C06321=1171.550,195.778,-60.007,-177.951,6.897,148.679
C06322=1171.554,195.530,-59.983,-177.954,6.895,148.679
C06323=1171.559,195.280,-59.960,-177.956,6.893,148.680
C06324=1171.563,195.031,-59.937,-177.959,6.891,148.680
C06325=1171.568,194.783,-59.912,-177.962,6.889,148.680
C06326=1171.572,194.534,-59.889,-177.964,6.887,148.681
C06327=1171.577,194.285,-59.866,-177.967,6.885,148.681
C06328=1171.582,194.037,-59.842,-177.970,6.882,148.681
C06329=1171.586,193.788,-59.818,-177.973,6.881,148.682
C06330=1171.591,193.539,-59.795,-177.975,6.879,148.682
C06331=1171.595,193.290,-59.771,-177.978,6.876,148.682
C06332=1171.600,193.041,-59.748,-177.981,6.874,148.682
C06333=1171.605,192.792,-59.724,-177.983,6.872,148.682
C06334=1171.609,192.544,-59.700,-177.986,6.870,148.683
C06335=1171.614,192.295,-59.677,-177.989,6.868,148.683
C06336=1171.619,192.046,-59.653,-177.992,6.866,148.684
C06337=1171.623,191.797,-59.630,-177.994,6.864,148.684
C06338=1171.628,191.547,-59.607,-177.997,6.862,148.684
C06339=1171.632,191.299,-59.583,-178.000,6.859,148.684
C06340=1171.637,191.050,-59.559,-178.003,6.858,148.685
C06341=1171.642,190.801,-59.536,-178.005,6.856,148.685
C06342=1171.646,190.552,-59.513,-178.007,6.854,148.685
C06343=1171.652,190.304,-59.490,-178.011,6.851,148.685
C06344=1171.656,190.055,-59.467,-178.013,6.849,148.686
C06345=1171.660,189.807,-59.443,-178.016,6.847,148.686
C06346=1171.665,189.557,-59.419,-178.018,6.845,148.686
C06347=1171.669,189.308,-59.396,-178.022,6.843,148.687
C06348=1171.674,189.059,-59.373,-178.024,6.841,148.687
C06349=1171.679,188.810,-59.349,-178.026,6.839,148.687
C06350=1171.684,188.561,-59.326,-178.029,6.837,148.688
C06351=1171.688,188.313,-59.303,-178.032,6.835,148.688
C06352=1171.692,188.064,-59.280,-178.035,6.833,148.688
C06353=1171.697,187.815,-59.256,-178.038,6.831,148.689
C06354=1171.702,187.566,-59.233,-178.040,6.829,148.689
C06355=1171.707,187.317,-59.210,-178.043,6.826,148.689
C06356=1171.711,187.068,-59.187,-178.046,6.825,148.689
C06357=1171.716,186.819,-59.164,-178.049,6.823,148.690
C06358=1171.720,186.570,-59.141,-178.051,6.821,148.690
C06359=1171.725,186.321,-59.117,-178.053,6.819,148.690
C06360=1171.729,186.073,-59.094,-178.057,6.816,148.691
C06361=1171.734,185.824,-59.071,-178.059,6.815,148.691
C06362=1171.739,185.575,-59.048,-178.062,6.813,148.691
C06363=1171.744,185.326,-59.025,-178.064,6.811,148.691
C06364=1171.748,185.078,-59.002,-178.067,6.808,148.692
C06365=1171.752,184.829,-58.979,-178.070,6.806,148.692
C06366=1171.758,184.559,-58.954,-178.073,6.805,148.692
C06367=1171.762,184.289,-58.929,-178.076,6.802,148.693
C06368=1171.768,184.020,-58.904,-178.079,6.800,148.693
C06369=1171.773,183.750,-58.879,-178.082,6.798,148.693
C06370=1171.777,183.501,-58.856,-178.085,6.796,148.694
C06371=1171.782,183.252,-58.833,-178.087,6.794,148.694
C06372=1171.786,183.003,-58.810,-178.090,6.792,148.694
C06373=1171.791,182.754,-58.788,-178.092,6.790,148.695
C06374=1171.796,182.505,-58.765,-178.095,6.788,148.695
C06375=1171.800,182.256,-58.741,-178.098,6.786,148.695
C06376=1171.804,182.008,-58.718,-178.100,6.784,148.696
C06377=1171.810,181.759,-58.696,-178.103,6.782,148.696
C06378=1171.814,181.510,-58.673,-178.106,6.780,148.696
C06379=1171.819,181.261,-58.650,-178.109,6.778,148.697
C06380=1171.823,181.012,-58.627,-178.112,6.776,148.697
C06381=1171.828,180.762,-58.605,-178.114,6.774,148.697
C06382=1171.833,180.514,-58.582,-178.117,6.772,148.697
C06383=1171.837,180.265,-58.559,-178.119,6.770,148.698
C06384=1171.842,180.016,-58.536,-178.122,6.768,148.698
C06385=1171.846,179.767,-58.513,-178.125,6.766,148.698
C06386=1171.851,179.519,-58.490,-178.128,6.764,148.699
C06387=1171.855,179.269,-58.468,-178.131,6.762,148.699
C06388=1171.860,179.020,-58.445,-178.133,6.760,148.699
C06389=1171.865,178.772,-58.423,-178.135,6.758,148.700
C06390=1171.870,178.523,-58.400,-178.139,6.756,148.700
C06391=1171.874,178.274,-58.377,-178.141,6.754,148.700
C06392=1171.879,178.024,-58.355,-178.144,6.752,148.701
C06393=1171.883,177.776,-58.332,-178.147,6.750,148.701
C06394=1171.888,177.527,-58.310,-178.149,6.748,148.701
C06395=1171.892,177.278,-58.287,-178.152,6.747,148.702
C06396=1171.898,177.030,-58.264,-178.155,6.744,148.702
C06397=1171.902,176.780,-58.242,-178.158,6.742,148.702
C06398=1171.907,176.531,-58.218,-178.160,6.740,148.703
C06399=1171.911,176.283,-58.197,-178.163,6.739,148.703
C06400=1171.916,176.034,-58.173,-178.166,6.737,148.703
C06401=1171.920,175.784,-58.151,-178.168,6.735,148.704
C06402=1171.925,175.536,-58.129,-178.170,6.733,148.704
C06403=1171.930,175.287,-58.106,-178.174,6.730,148.704
C06404=1171.934,175.037,-58.084,-178.176,6.729,148.705
C06405=1171.940,174.789,-58.061,-178.179,6.727,148.705
C06406=1171.944,174.539,-58.039,-178.182,6.725,148.705
C06407=1171.948,174.291,-58.016,-178.184,6.723,148.706
C06408=1171.953,174.042,-57.994,-178.187,6.722,148.706
C06409=1171.958,173.792,-57.972,-178.189,6.720,148.706
C06410=1171.963,173.544,-57.949,-178.193,6.717,148.707
C06411=1171.967,173.295,-57.927,-178.195,6.715,148.707
C06412=1171.971,173.046,-57.904,-178.198,6.713,148.707
C06413=1171.977,172.797,-57.882,-178.201,6.712,148.708
C06414=1171.981,172.548,-57.860,-178.203,6.710,148.708
C06415=1171.986,172.300,-57.838,-178.206,6.708,148.708
C06416=1171.991,172.050,-57.815,-178.209,6.706,148.709
C06417=1171.995,171.801,-57.793,-178.211,6.705,148.709
C06418=1172.000,171.552,-57.771,-178.214,6.702,148.709
C06419=1172.004,171.303,-57.748,-178.217,6.700,148.710
C06420=1172.009,171.054,-57.726,-178.220,6.698,148.710
C06421=1172.014,170.805,-57.704,-178.222,6.696,148.710
C06422=1172.018,170.556,-57.682,-178.225,6.695,148.711
C06423=1172.023,170.307,-57.659,-178.228,6.693,148.711
C06424=1172.028,170.059,-57.637,-178.230,6.691,148.711
C06425=1172.032,169.809,-57.615,-178.233,6.689,148.712
C06426=1172.037,169.560,-57.593,-178.236,6.688,148.712
C06427=1172.042,169.311,-57.571,-178.239,6.685,148.713
C06428=1172.046,169.062,-57.548,-178.242,6.683,148.713
C06429=1172.051,168.814,-57.527,-178.244,6.681,148.713
C06430=1172.055,168.564,-57.505,-178.246,6.679,148.713
C06431=1172.060,168.316,-57.483,-178.249,6.678,148.714
C06432=1172.065,168.066,-57.460,-178.252,6.676,148.714
C06433=1172.070,167.818,-57.438,-178.255,6.674,148.715
C06434=1172.074,167.568,-57.416,-178.257,6.672,148.715
C06435=1172.079,167.320,-57.395,-178.260,6.671,148.715
C06436=1172.083,167.070,-57.373,-178.263,6.669,148.716
C06437=1172.089,166.822,-57.350,-178.265,6.667,148.716
C06438=1172.093,166.573,-57.328,-178.269,6.664,148.716
C06439=1172.098,166.324,-57.306,-178.271,6.663,148.717
C06440=1172.102,166.075,-57.284,-178.274,6.661,148.717
C06441=1172.107,165.826,-57.262,-178.277,6.659,148.717
C06442=1172.111,165.577,-57.240,-178.279,6.657,148.718
C06443=1172.116,165.328,-57.219,-178.281,6.655,148.718
C06444=1172.121,165.079,-57.197,-178.284,6.654,148.718
C06445=1172.125,164.830,-57.175,-178.287,6.652,148.719
C06446=1172.131,164.581,-57.153,-178.290,6.650,148.719
C06447=1172.135,164.332,-57.130,-178.292,6.648,148.719
C06448=1172.140,164.083,-57.109,-178.295,6.647,148.720
C06449=1172.144,163.834,-57.087,-178.298,6.645,148.720
C06450=1172.149,163.584,-57.066,-178.300,6.643,148.721
C06451=1172.154,163.336,-57.044,-178.303,6.641,148.721
C06452=1172.159,163.086,-57.022,-178.306,6.640,148.721
C06453=1172.163,162.838,-57.000,-178.309,6.637,148.722
C06454=1172.168,162.588,-56.978,-178.312,6.635,148.722
C06455=1172.173,162.340,-56.957,-178.314,6.633,148.722
C06456=1172.177,162.090,-56.935,-178.317,6.632,148.723
C06457=1172.182,161.842,-56.913,-178.320,6.630,148.723
C06458=1172.187,161.593,-56.892,-178.322,6.628,148.724
C06459=1172.191,161.343,-56.870,-178.325,6.626,148.724
C06460=1172.196,161.095,-56.848,-178.328,6.625,148.724
C06461=1172.201,160.846,-56.827,-178.330,6.623,148.725
C06462=1172.205,160.597,-56.804,-178.333,6.621,148.725
C06463=1172.210,160.347,-56.784,-178.336,6.619,148.725
C06464=1172.215,160.098,-56.761,-178.339,6.618,148.726
C06465=1172.219,159.849,-56.740,-178.341,6.616,148.726
C06466=1172.224,159.601,-56.718,-178.344,6.614,148.727
C06467=1172.229,159.351,-56.697,-178.347,6.612,148.727
C06468=1172.233,159.102,-56.676,-178.349,6.611,148.727
C06469=1172.238,158.854,-56.654,-178.352,6.609,148.728
C06470=1172.243,158.584,-56.631,-178.355,6.607,148.728
C06471=1172.248,158.315,-56.608,-178.358,6.604,148.728
C06472=1172.253,158.047,-56.584,-178.361,6.603,148.729
C06473=1172.258,157.778,-56.561,-178.363,6.601,148.729
C06474=1172.263,157.529,-56.539,-178.366,6.599,148.730
C06475=1172.268,157.279,-56.518,-178.369,6.597,148.730
C06476=1172.272,157.030,-56.496,-178.371,6.596,148.730
C06477=1172.278,156.781,-56.475,-178.374,6.594,148.731
C06478=1172.282,156.532,-56.454,-178.377,6.592,148.731
C06479=1172.286,156.283,-56.432,-178.379,6.590,148.731
C06480=1172.291,156.034,-56.411,-178.382,6.589,148.732
C06481=1172.296,155.786,-56.390,-178.385,6.587,148.732
C06482=1172.301,155.536,-56.369,-178.388,6.585,148.733
C06483=1172.305,155.287,-56.347,-178.390,6.583,148.733
C06484=1172.311,155.038,-56.326,-178.393,6.582,148.733
C06485=1172.315,154.789,-56.305,-178.396,6.580,148.734
C06486=1172.319,154.540,-56.282,-178.398,6.578,148.734
C06487=1172.324,154.291,-56.262,-178.401,6.576,148.734
C06488=1172.329,154.042,-56.240,-178.404,6.575,148.735
C06489=1172.333,153.793,-56.219,-178.406,6.573,148.735
C06490=1172.339,153.544,-56.198,-178.409,6.571,148.736
C06491=1172.343,153.295,-56.176,-178.412,6.569,148.736
C06492=1172.348,153.045,-56.155,-178.414,6.568,148.736
C06493=1172.352,152.797,-56.134,-178.417,6.566,148.737
C06494=1172.357,152.548,-56.113,-178.420,6.564,148.737
C06495=1172.362,152.298,-56.091,-178.423,6.562,148.737
C06496=1172.367,152.049,-56.070,-178.426,6.561,148.738
C06497=1172.371,151.800,-56.050,-178.428,6.559,148.738
C06498=1172.376,151.552,-56.028,-178.431,6.558,148.739
C06499=1172.381,151.302,-56.007,-178.434,6.556,148.739
C06500=1172.385,151.054,-55.986,-178.436,6.554,148.740
C06501=1172.390,150.804,-55.965,-178.439,6.552,148.740
C06502=1172.395,150.555,-55.944,-178.442,6.551,148.740
C06503=1172.399,150.306,-55.923,-178.445,6.549,148.741
C06504=1172.405,150.057,-55.902,-178.447,6.547,148.741
C06505=1172.410,149.808,-55.881,-178.450,6.545,148.741
C06506=1172.414,149.559,-55.861,-178.453,6.544,148.742
C06507=1172.418,149.310,-55.839,-178.455,6.542,148.742
C06508=1172.424,149.060,-55.818,-178.458,6.540,148.743
C06509=1172.428,148.811,-55.797,-178.461,6.538,148.743
C06510=1172.433,148.563,-55.776,-178.463,6.537,148.743
C06511=1172.437,148.314,-55.755,-178.466,6.535,148.744
C06512=1172.443,148.065,-55.734,-178.469,6.533,148.744
C06513=1172.448,147.815,-55.713,-178.472,6.531,148.744
C06514=1172.452,147.566,-55.693,-178.474,6.530,148.745
C06515=1172.456,147.317,-55.671,-178.477,6.529,148.745
C06516=1172.461,147.068,-55.650,-178.479,6.527,148.746
C06517=1172.466,146.819,-55.629,-178.482,6.525,148.746
C06518=1172.470,146.570,-55.609,-178.485,6.524,148.747
C06519=1172.476,146.321,-55.588,-178.488,6.522,148.747
C06520=1172.480,146.072,-55.568,-178.490,6.520,148.747
C06521=1172.485,145.823,-55.546,-178.493,6.518,148.748
C06522=1172.489,145.574,-55.526,-178.496,6.517,148.748
C06523=1172.495,145.325,-55.505,-178.498,6.515,148.749
C06524=1172.499,145.076,-55.484,-178.501,6.513,148.749
C06525=1172.504,144.827,-55.463,-178.504,6.511,148.749
C06526=1172.508,144.577,-55.443,-178.506,6.510,148.750
C06527=1172.513,144.328,-55.422,-178.509,6.508,148.750
C06528=1172.518,144.079,-55.401,-178.512,6.507,148.751
C06529=1172.523,143.829,-55.380,-178.515,6.505,148.751
C06530=1172.527,143.580,-55.360,-178.517,6.504,148.751
C06531=1172.532,143.331,-55.339,-178.520,6.502,148.752
C06532=1172.537,143.082,-55.319,-178.523,6.500,148.752
C06533=1172.542,142.833,-55.298,-178.525,6.499,148.753
C06534=1172.546,142.584,-55.277,-178.528,6.497,148.753
C06535=1172.551,142.335,-55.257,-178.531,6.495,148.753
C06536=1172.556,142.086,-55.236,-178.533,6.493,148.754
C06537=1172.560,141.837,-55.216,-178.536,6.492,148.754
C06538=1172.566,141.588,-55.195,-178.539,6.490,148.755
C06539=1172.570,141.339,-55.174,-178.542,6.489,148.755
C06540=1172.575,141.090,-55.154,-178.545,6.487,148.756
C06541=1172.580,140.840,-55.133,-178.547,6.486,148.756
C06542=1172.584,140.592,-55.113,-178.549,6.484,148.756
C06543=1172.589,140.343,-55.092,-178.552,6.482,148.757
C06544=1172.594,140.093,-55.071,-178.555,6.481,148.757
C06545=1172.598,139.844,-55.051,-178.558,6.479,148.758
C06546=1172.604,139.595,-55.031,-178.560,6.477,148.758
C06547=1172.608,139.346,-55.010,-178.563,6.476,148.758
C06548=1172.613,139.097,-54.990,-178.566,6.474,148.759
C06549=1172.617,138.848,-54.969,-178.569,6.472,148.759
C06550=1172.622,138.598,-54.948,-178.571,6.471,148.760
C06551=1172.627,138.349,-54.928,-178.574,6.470,148.760
C06552=1172.631,138.100,-54.908,-178.576,6.468,148.760
C06553=1172.637,137.851,-54.888,-178.579,6.466,148.761
C06554=1172.642,137.602,-54.867,-178.582,6.464,148.761
C06555=1172.646,137.353,-54.847,-178.585,6.463,148.762
C06556=1172.651,137.104,-54.827,-178.588,6.461,148.762
C06557=1172.656,136.855,-54.806,-178.590,6.460,148.763
C06558=1172.660,136.606,-54.786,-178.592,6.459,148.763
C06559=1172.665,136.357,-54.766,-178.595,6.457,148.763
C06560=1172.670,136.107,-54.746,-178.598,6.455,148.764
C06561=1172.675,135.858,-54.725,-178.601,6.453,148.764
C06562=1172.679,135.609,-54.705,-178.604,6.452,148.765
C06563=1172.684,135.359,-54.685,-178.606,6.450,148.765
C06564=1172.689,135.111,-54.665,-178.609,6.448,148.766
C06565=1172.694,134.862,-54.644,-178.612,6.447,148.766
C06566=1172.699,134.612,-54.624,-178.614,6.446,148.766
C06567=1172.703,134.363,-54.604,-178.617,6.444,148.767
C06568=1172.708,134.114,-54.584,-178.619,6.442,148.767
C06569=1172.712,133.865,-54.564,-178.622,6.441,148.768
C06570=1172.717,133.616,-54.544,-178.625,6.439,148.768
C06571=1172.723,133.367,-54.524,-178.628,6.437,148.769
C06572=1172.727,133.118,-54.503,-178.630,6.437,148.769
C06573=1172.732,132.869,-54.483,-178.633,6.435,148.769
C06574=1172.737,132.600,-54.462,-178.636,6.433,148.770
C06575=1172.742,132.331,-54.440,-178.639,6.432,148.770
C06576=1172.747,132.063,-54.419,-178.642,6.429,148.771
C06577=1172.753,131.794,-54.397,-178.645,6.428,148.771
C06578=1172.757,131.545,-54.376,-178.647,6.427,148.772
C06579=1172.762,131.296,-54.357,-178.650,6.425,148.772
C06580=1172.766,131.047,-54.336,-178.653,6.423,148.773
C06581=1172.772,130.798,-54.317,-178.655,6.422,148.773
C06582=1172.776,130.549,-54.297,-178.658,6.420,148.773
C06583=1172.781,130.299,-54.277,-178.661,6.419,148.774
C06584=1172.786,130.050,-54.257,-178.663,6.418,148.774
C06585=1172.790,129.801,-54.237,-178.666,6.416,148.775
C06586=1172.796,129.552,-54.217,-178.669,6.414,148.775
C06587=1172.801,129.303,-54.197,-178.671,6.412,148.776
C06588=1172.805,129.053,-54.177,-178.674,6.411,148.776
C06589=1172.810,128.804,-54.157,-178.677,6.410,148.777
C06590=1172.815,128.555,-54.137,-178.679,6.408,148.777
C06591=1172.820,128.306,-54.118,-178.682,6.407,148.777
C06592=1172.824,128.057,-54.097,-178.685,6.405,148.778
C06593=1172.829,127.807,-54.078,-178.688,6.403,148.778
C06594=1172.834,127.558,-54.059,-178.691,6.402,148.779
C06595=1172.839,127.309,-54.038,-178.693,6.401,148.779
C06596=1172.843,127.060,-54.018,-178.696,6.399,148.780
C06597=1172.848,126.810,-53.999,-178.698,6.397,148.780
C06598=1172.853,126.562,-53.979,-178.701,6.396,148.780
C06599=1172.857,126.313,-53.960,-178.704,6.394,148.781
C06600=1172.862,126.063,-53.940,-178.706,6.393,148.781
C06601=1172.866,125.814,-53.920,-178.709,6.392,148.782
C06602=1172.872,125.565,-53.900,-178.712,6.390,148.782
C06603=1172.877,125.316,-53.881,-178.714,6.388,148.783
C06604=1172.881,125.066,-53.861,-178.718,6.387,148.783
C06605=1172.886,124.818,-53.841,-178.720,6.386,148.784
C06606=1172.891,124.568,-53.821,-178.722,6.384,148.784
C06607=1172.896,124.319,-53.802,-178.725,6.382,148.784
C06608=1172.901,124.070,-53.783,-178.728,6.381,148.785
C06609=1172.905,123.821,-53.763,-178.730,6.380,148.785
C06610=1172.910,123.572,-53.743,-178.733,6.378,148.786
C06611=1172.915,123.323,-53.724,-178.736,6.377,148.786
C06612=1172.920,123.073,-53.704,-178.739,6.375,148.787
C06613=1172.924,122.824,-53.684,-178.742,6.373,148.787
C06614=1172.930,122.575,-53.665,-178.744,6.373,148.788
C06615=1172.934,122.325,-53.646,-178.747,6.371,148.788
C06616=1172.939,122.076,-53.626,-178.749,6.369,148.788
C06617=1172.944,121.827,-53.607,-178.752,6.367,148.789
C06618=1172.948,121.578,-53.587,-178.755,6.367,148.789
C06619=1172.953,121.329,-53.567,-178.757,6.365,148.790
C06620=1172.958,121.080,-53.548,-178.760,6.363,148.790
C06621=1172.962,120.831,-53.529,-178.763,6.362,148.791
C06622=1172.968,120.582,-53.510,-178.765,6.361,148.791
C06623=1172.972,120.332,-53.490,-178.768,6.359,148.792
C06624=1172.977,120.083,-53.470,-178.771,6.358,148.792
C06625=1172.983,119.834,-53.451,-178.773,6.356,148.792
C06626=1172.987,119.584,-53.432,-178.776,6.355,148.793
C06627=1172.992,119.336,-53.413,-178.779,6.354,148.794
C06628=1172.997,119.086,-53.393,-178.782,6.352,148.794
C06629=1173.001,118.836,-53.373,-178.784,6.350,148.794
C06630=1173.006,118.588,-53.355,-178.787,6.350,148.795
C06631=1173.011,118.338,-53.335,-178.790,6.348,148.795
C06632=1173.016,118.089,-53.316,-178.792,6.346,148.796
C06633=1173.020,117.840,-53.297,-178.795,6.344,148.796
C06634=1173.025,117.591,-53.277,-178.798,6.344,148.797
C06635=1173.030,117.342,-53.258,-178.800,6.342,148.797
C06636=1173.036,117.092,-53.239,-178.803,6.340,148.798
C06637=1173.040,116.843,-53.220,-178.806,6.339,148.798
C06638=1173.045,116.593,-53.200,-178.808,6.338,148.799
C06639=1173.050,116.345,-53.181,-178.811,6.336,148.799
C06640=1173.054,116.095,-53.162,-178.814,6.335,148.799
C06641=1173.059,115.846,-53.143,-178.816,6.333,148.800
C06642=1173.064,115.597,-53.123,-178.819,6.332,148.800
C06643=1173.069,115.348,-53.104,-178.822,6.331,148.801
C06644=1173.074,115.098,-53.085,-178.824,6.329,148.801
C06645=1173.078,114.850,-53.067,-178.827,6.328,148.802
C06646=1173.083,114.600,-53.047,-178.830,6.327,148.802
C06647=1173.088,114.351,-53.028,-178.832,6.325,148.803
C06648=1173.092,114.102,-53.009,-178.835,6.323,148.803
C06649=1173.098,113.852,-52.990,-178.838,6.323,148.804
C06650=1173.102,113.603,-52.971,-178.841,6.321,148.804
C06651=1173.107,113.354,-52.952,-178.843,6.319,148.805
C06652=1173.112,113.105,-52.932,-178.845,6.318,148.805
C06653=1173.117,112.856,-52.914,-178.849,6.317,148.806
C06654=1173.122,112.606,-52.894,-178.851,6.315,148.806
C06655=1173.126,112.357,-52.876,-178.854,6.313,148.806
C06656=1173.132,112.108,-52.857,-178.856,6.312,148.807
C06657=1173.136,111.859,-52.838,-178.859,6.311,148.807
C06658=1173.141,111.610,-52.819,-178.862,6.309,148.808
C06659=1173.146,111.360,-52.800,-178.864,6.308,148.808
C06660=1173.151,111.111,-52.781,-178.867,6.307,148.809
C06661=1173.156,110.861,-52.762,-178.870,6.305,148.809
C06662=1173.161,110.612,-52.744,-178.872,6.304,148.810
C06663=1173.166,110.363,-52.724,-178.875,6.303,148.810
C06664=1173.170,110.114,-52.705,-178.878,6.301,148.811
C06665=1173.176,109.865,-52.687,-178.880,6.300,148.811
C06666=1173.180,109.615,-52.668,-178.883,6.299,148.812
C06667=1173.185,109.366,-52.650,-178.886,6.297,148.812
C06668=1173.189,109.117,-52.630,-178.889,6.296,148.813
C06669=1173.194,108.868,-52.611,-178.891,6.295,148.813
C06670=1173.200,108.619,-52.593,-178.894,6.293,148.814
C06671=1173.204,108.369,-52.574,-178.897,6.292,148.814
C06672=1173.209,108.120,-52.555,-178.899,6.291,148.814
C06673=1173.213,107.871,-52.536,-178.902,6.289,148.815
C06674=1173.219,107.621,-52.517,-178.905,6.288,148.816
C06675=1173.223,107.373,-52.499,-178.907,6.287,148.816
C06676=1173.228,107.123,-52.480,-178.910,6.285,148.816
C06677=1173.233,106.874,-52.461,-178.913,6.284,148.817
C06678=1173.238,106.606,-52.442,-178.915,6.283,148.817
C06679=1173.243,106.337,-52.421,-178.918,6.281,148.818
C06680=1173.248,106.069,-52.401,-178.921,6.280,148.818
C06681=1173.254,105.800,-52.381,-178.924,6.278,148.819
C06682=1173.259,105.552,-52.362,-178.927,6.277,148.819
C06683=1173.264,105.301,-52.344,-178.929,6.276,148.820
C06684=1173.269,105.052,-52.326,-178.932,6.274,148.821
C06685=1173.273,104.804,-52.307,-178.935,6.273,148.821
C06686=1173.278,104.553,-52.288,-178.937,6.272,148.821
C06687=1173.283,104.305,-52.269,-178.940,6.270,148.822
C06688=1173.288,104.056,-52.251,-178.943,6.269,148.822
C06689=1173.293,103.806,-52.232,-178.945,6.268,148.823
C06690=1173.297,103.557,-52.214,-178.948,6.266,148.823
C06691=1173.302,103.308,-52.196,-178.951,6.265,148.824
C06692=1173.307,103.058,-52.177,-178.953,6.264,148.824
C06693=1173.312,102.809,-52.158,-178.956,6.262,148.825
C06694=1173.317,102.560,-52.140,-178.959,6.261,148.825
C06695=1173.322,102.311,-52.122,-178.961,6.260,148.826
C06696=1173.327,102.061,-52.102,-178.964,6.258,148.826
C06697=1173.331,101.812,-52.084,-178.967,6.258,148.827
C06698=1173.336,101.563,-52.066,-178.969,6.256,148.827
C06699=1173.341,101.313,-52.048,-178.973,6.254,148.828
C06700=1173.346,101.064,-52.029,-178.975,6.254,148.828
C06701=1173.351,100.815,-52.011,-178.977,6.252,148.829
C06702=1173.356,100.566,-51.993,-178.981,6.250,148.829
C06703=1173.360,100.316,-51.974,-178.983,6.250,148.830
C06704=1173.366,100.067,-51.955,-178.985,6.248,148.830
C06705=1173.370,99.818,-51.937,-178.988,6.247,148.831
C06706=1173.375,99.569,-51.919,-178.991,6.246,148.831
C06707=1173.380,99.319,-51.901,-178.993,6.244,148.832
C06708=1173.385,99.070,-51.883,-178.996,6.243,148.832
C06709=1173.389,98.821,-51.864,-178.999,6.242,148.833
C06710=1173.395,98.572,-51.846,-179.001,6.241,148.833
C06711=1173.400,98.322,-51.828,-179.004,6.239,148.834
C06712=1173.404,98.072,-51.809,-179.007,6.238,148.834
C06713=1173.409,97.823,-51.791,-179.009,6.237,148.835
C06714=1173.414,97.574,-51.773,-179.012,6.235,148.835
C06715=1173.419,97.325,-51.755,-179.014,6.234,148.836
C06716=1173.424,97.075,-51.737,-179.018,6.233,148.836
C06717=1173.429,96.826,-51.719,-179.020,6.231,148.837
C06718=1173.434,96.576,-51.700,-179.022,6.230,148.837
C06719=1173.438,96.328,-51.682,-179.026,6.229,148.838
C06720=1173.443,96.079,-51.664,-179.028,6.228,148.838
C06721=1173.448,95.830,-51.646,-179.030,6.227,148.839
C06722=1173.453,95.580,-51.628,-179.034,6.225,148.839
C06723=1173.458,95.331,-51.610,-179.036,6.224,148.840
C06724=1173.462,95.081,-51.591,-179.039,6.223,148.840
C06725=1173.467,94.832,-51.574,-179.041,6.222,148.841
C06726=1173.472,94.583,-51.556,-179.044,6.220,148.841
C06727=1173.477,94.334,-51.538,-179.047,6.219,148.842
C06728=1173.483,94.084,-51.519,-179.049,6.218,148.842
C06729=1173.488,93.835,-51.501,-179.052,6.216,148.843
C06730=1173.492,93.586,-51.483,-179.055,6.216,148.843
C06731=1173.497,93.335,-51.465,-179.057,6.214,148.844
C06732=1173.502,93.086,-51.447,-179.060,6.214,148.844
C06733=1173.507,92.837,-51.429,-179.063,6.212,148.845
C06734=1173.512,92.588,-51.411,-179.065,6.210,148.845
C06735=1173.517,92.339,-51.393,-179.068,6.210,148.846
C06736=1173.522,92.090,-51.375,-179.071,6.208,148.846
C06737=1173.527,91.840,-51.358,-179.073,6.207,148.847
C06738=1173.531,91.591,-51.340,-179.076,6.206,148.847
C06739=1173.536,91.342,-51.322,-179.078,6.205,148.848
C06740=1173.541,91.093,-51.304,-179.081,6.203,148.848
C06741=1173.545,90.843,-51.287,-179.084,6.202,148.849
C06742=1173.550,90.593,-51.269,-179.087,6.201,148.849
C06743=1173.555,90.344,-51.251,-179.089,6.199,148.850
C06744=1173.560,90.095,-51.233,-179.092,6.199,148.850
C06745=1173.565,89.846,-51.215,-179.095,6.197,148.851
C06746=1173.570,89.596,-51.197,-179.097,6.196,148.851
C06747=1173.575,89.347,-51.179,-179.100,6.195,148.852
C06748=1173.580,89.098,-51.161,-179.102,6.194,148.852
C06749=1173.585,88.849,-51.143,-179.105,6.192,148.853
C06750=1173.590,88.599,-51.126,-179.108,6.192,148.853
C06751=1173.595,88.350,-51.108,-179.110,6.190,148.854
C06752=1173.599,88.101,-51.091,-179.114,6.189,148.854
C06753=1173.604,87.852,-51.073,-179.116,6.188,148.855
C06754=1173.609,87.602,-51.056,-179.118,6.186,148.855
C06755=1173.614,87.353,-51.038,-179.121,6.186,148.856
C06756=1173.619,87.103,-51.020,-179.124,6.184,148.856
C06757=1173.624,86.854,-51.002,-179.126,6.183,148.857
C06758=1173.629,86.605,-50.984,-179.129,6.182,148.857
C06759=1173.633,86.356,-50.967,-179.131,6.181,148.858
C06760=1173.639,86.106,-50.950,-179.134,6.179,148.859
C06761=1173.643,85.857,-50.932,-179.137,6.179,148.859
C06762=1173.648,85.608,-50.914,-179.140,6.177,148.860
C06763=1173.654,85.358,-50.896,-179.142,6.176,148.860
C06764=1173.658,85.109,-50.878,-179.145,6.175,148.860
C06765=1173.663,84.860,-50.861,-179.147,6.174,148.861
C06766=1173.668,84.610,-50.844,-179.150,6.172,148.862
C06767=1173.673,84.361,-50.826,-179.153,6.172,148.862
C06768=1173.678,84.111,-50.809,-179.155,6.170,148.863
C06769=1173.682,83.862,-50.791,-179.159,6.169,148.863
C06770=1173.687,83.612,-50.774,-179.161,6.168,148.864
C06771=1173.692,83.363,-50.756,-179.163,6.166,148.864
C06772=1173.697,83.114,-50.738,-179.166,6.166,148.865
C06773=1173.702,82.864,-50.721,-179.169,6.164,148.865
C06774=1173.707,82.615,-50.703,-179.171,6.163,148.866
C06775=1173.712,82.366,-50.686,-179.174,6.162,148.866
C06776=1173.717,82.117,-50.668,-179.177,6.161,148.867
C06777=1173.722,81.867,-50.652,-179.179,6.159,148.867
C06778=1173.727,81.618,-50.634,-179.182,6.159,148.868
C06779=1173.732,81.369,-50.617,-179.185,6.157,148.868
C06780=1173.736,81.120,-50.599,-179.187,6.156,148.869
C06781=1173.741,80.870,-50.582,-179.190,6.155,148.869
C06782=1173.747,80.601,-50.563,-179.192,6.154,148.870
C06783=1173.752,80.333,-50.544,-179.196,6.153,148.871
C06784=1173.757,80.065,-50.526,-179.199,6.151,148.871
C06785=1173.762,79.796,-50.507,-179.201,6.151,148.872
C06786=1173.767,79.547,-50.489,-179.204,6.149,148.872
C06787=1173.772,79.298,-50.473,-179.206,6.148,148.873
C06788=1173.778,79.048,-50.456,-179.209,6.147,148.873
C06789=1173.783,78.799,-50.438,-179.212,6.146,148.874
C06790=1173.787,78.550,-50.421,-179.215,6.145,148.874
C06791=1173.792,78.300,-50.404,-179.217,6.144,148.875
C06792=1173.796,78.051,-50.387,-179.220,6.142,148.875
C06793=1173.802,77.801,-50.369,-179.222,6.142,148.876
C06794=1173.807,77.552,-50.352,-179.225,6.140,148.876
C06795=1173.812,77.303,-50.335,-179.228,6.139,148.877
C06796=1173.817,77.053,-50.318,-179.230,6.138,148.877
C06797=1173.821,76.804,-50.301,-179.233,6.137,148.878
C06798=1173.826,76.555,-50.283,-179.235,6.136,148.879
C06799=1173.831,76.305,-50.266,-179.238,6.135,148.879
C06800=1173.837,76.056,-50.249,-179.241,6.134,148.880
C06801=1173.842,75.806,-50.232,-179.244,6.133,148.880
C06802=1173.846,75.557,-50.215,-179.246,6.132,148.881
C06803=1173.851,75.308,-50.198,-179.249,6.130,148.881
C06804=1173.856,75.058,-50.181,-179.251,6.130,148.882
C06805=1173.861,74.809,-50.164,-179.254,6.128,148.882
C06806=1173.866,74.560,-50.147,-179.257,6.127,148.883
C06807=1173.871,74.310,-50.129,-179.259,6.126,148.883
C06808=1173.875,74.061,-50.113,-179.262,6.125,148.884
C06809=1173.881,73.811,-50.095,-179.264,6.124,148.884
C06810=1173.886,73.562,-50.079,-179.267,6.123,148.885
C06811=1173.891,73.313,-50.062,-179.269,6.122,148.885
C06812=1173.895,73.064,-50.044,-179.273,6.121,148.886
C06813=1173.900,72.814,-50.027,-179.275,6.120,148.887
C06814=1173.905,72.565,-50.011,-179.278,6.119,148.887
C06815=1173.911,72.315,-49.994,-179.280,6.118,148.888
C06816=1173.915,72.066,-49.977,-179.283,6.116,148.888
C06817=1173.920,71.816,-49.960,-179.286,6.115,148.889
C06818=1173.925,71.567,-49.943,-179.288,6.115,148.889
C06819=1173.930,71.318,-49.927,-179.291,6.113,148.890
C06820=1173.935,71.068,-49.909,-179.293,6.112,148.890
C06821=1173.940,70.819,-49.893,-179.296,6.111,148.891
C06822=1173.945,70.569,-49.876,-179.298,6.110,148.891
C06823=1173.950,70.321,-49.859,-179.302,6.109,148.892
C06824=1173.954,70.071,-49.842,-179.304,6.108,148.892
C06825=1173.960,69.822,-49.825,-179.306,6.107,148.893
C06826=1173.964,69.572,-49.808,-179.309,6.106,148.894
C06827=1173.970,69.323,-49.791,-179.312,6.105,148.894
C06828=1173.974,69.073,-49.774,-179.314,6.103,148.895
C06829=1173.979,68.824,-49.758,-179.317,6.103,148.895
C06830=1173.984,68.575,-49.741,-179.319,6.102,148.896
C06831=1173.989,68.325,-49.724,-179.322,6.101,148.896
C06832=1173.994,68.076,-49.708,-179.325,6.100,148.897
C06833=1173.999,67.826,-49.691,-179.328,6.098,148.897
C06834=1174.004,67.576,-49.675,-179.330,6.098,148.898
C06835=1174.009,67.328,-49.658,-179.333,6.096,148.899
C06836=1174.014,67.078,-49.641,-179.335,6.095,148.899
C06837=1174.019,66.828,-49.624,-179.338,6.095,148.900
C06838=1174.024,66.580,-49.608,-179.341,6.093,148.900
C06839=1174.029,66.330,-49.591,-179.343,6.093,148.901
C06840=1174.033,66.080,-49.574,-179.346,6.091,148.901
C06841=1174.038,65.832,-49.558,-179.349,6.090,148.902
C06842=1174.043,65.582,-49.541,-179.351,6.090,148.902
C06843=1174.049,65.332,-49.525,-179.354,6.088,148.903
C06844=1174.054,65.083,-49.508,-179.356,6.087,148.903
C06845=1174.058,64.833,-49.492,-179.359,6.086,148.904
C06846=1174.063,64.585,-49.475,-179.362,6.085,148.904
C06847=1174.068,64.335,-49.458,-179.364,6.085,148.905
C06848=1174.073,64.085,-49.441,-179.367,6.083,148.906
C06849=1174.078,63.836,-49.426,-179.370,6.082,148.906
C06850=1174.083,63.586,-49.409,-179.372,6.082,148.907
C06851=1174.089,63.337,-49.392,-179.375,6.080,148.907
C06852=1174.093,63.088,-49.376,-179.377,6.079,148.908
C06853=1174.098,62.838,-49.360,-179.380,6.078,148.908
C06854=1174.103,62.589,-49.343,-179.382,6.077,148.909
C06855=1174.107,62.339,-49.327,-179.385,6.077,148.910
C06856=1174.113,62.090,-49.310,-179.388,6.075,148.910
C06857=1174.118,61.840,-49.294,-179.390,6.074,148.911
C06858=1174.123,61.592,-49.277,-179.393,6.074,148.911
C06859=1174.128,61.342,-49.261,-179.396,6.072,148.912
C06860=1174.132,61.093,-49.244,-179.398,6.071,148.912
C06861=1174.137,60.843,-49.229,-179.401,6.070,148.913
C06862=1174.143,60.593,-49.211,-179.403,6.069,148.913
C06863=1174.148,60.345,-49.195,-179.406,6.069,148.914
C06864=1174.152,60.094,-49.179,-179.409,6.067,148.915
C06865=1174.158,59.846,-49.163,-179.411,6.066,148.915
C06866=1174.162,59.596,-49.147,-179.414,6.066,148.916
C06867=1174.167,59.347,-49.130,-179.417,6.064,148.916
C06868=1174.172,59.097,-49.114,-179.419,6.064,148.917
C06869=1174.177,58.848,-49.098,-179.422,6.063,148.917
C06870=1174.182,58.598,-49.082,-179.425,6.062,148.918
C06871=1174.188,58.349,-49.065,-179.427,6.061,148.918
C06872=1174.192,58.099,-49.049,-179.430,6.060,148.919
C06873=1174.197,57.850,-49.032,-179.432,6.058,148.919
C06874=1174.202,57.600,-49.016,-179.435,6.058,148.920
C06875=1174.207,57.352,-49.000,-179.438,6.056,148.920
C06876=1174.212,57.101,-48.984,-179.440,6.056,148.921
C06877=1174.217,56.853,-48.968,-179.442,6.055,148.922
C06878=1174.222,56.603,-48.952,-179.446,6.054,148.922
C06879=1174.227,56.354,-48.936,-179.448,6.053,148.923
C06880=1174.232,56.104,-48.920,-179.450,6.052,148.923
C06881=1174.237,55.855,-48.903,-179.454,6.051,148.924
C06882=1174.242,55.605,-48.887,-179.456,6.050,148.924
C06883=1174.247,55.356,-48.871,-179.458,6.049,148.925
C06884=1174.252,55.106,-48.855,-179.461,6.048,148.926
C06885=1174.257,54.857,-48.839,-179.464,6.047,148.926
C06886=1174.262,54.589,-48.822,-179.466,6.046,148.927
C06887=1174.267,54.319,-48.804,-179.469,6.045,148.927
C06888=1174.273,54.051,-48.787,-179.472,6.045,148.928
C06889=1174.278,53.783,-48.770,-179.475,6.043,148.929
C06890=1174.283,53.533,-48.754,-179.477,6.042,148.929
C06891=1174.288,53.284,-48.738,-179.480,6.041,148.930
C06892=1174.293,53.035,-48.722,-179.483,6.040,148.930
C06893=1174.298,52.785,-48.706,-179.485,6.040,148.931
C06894=1174.303,52.536,-48.690,-179.487,6.039,148.931
C06895=1174.308,52.286,-48.674,-179.491,6.037,148.932
C06896=1174.313,52.036,-48.658,-179.493,6.037,148.932
C06897=1174.318,51.788,-48.642,-179.495,6.036,148.933
C06898=1174.323,51.538,-48.626,-179.499,6.035,148.934
C06899=1174.329,51.288,-48.610,-179.501,6.034,148.934
C06900=1174.333,51.039,-48.594,-179.503,6.033,148.935
C06901=1174.338,50.789,-48.578,-179.506,6.032,148.935
C06902=1174.343,50.540,-48.563,-179.509,6.031,148.936
C06903=1174.348,50.291,-48.546,-179.511,6.030,148.936
C06904=1174.353,50.041,-48.531,-179.514,6.029,148.937
C06905=1174.358,49.791,-48.515,-179.516,6.028,148.938
C06906=1174.363,49.542,-48.499,-179.519,6.028,148.938
C06907=1174.368,49.293,-48.483,-179.521,6.027,148.939
C06908=1174.373,49.043,-48.467,-179.524,6.025,148.939
C06909=1174.378,48.794,-48.452,-179.527,6.025,148.940
C06910=1174.383,48.544,-48.436,-179.529,6.024,148.940
C06911=1174.387,48.295,-48.420,-179.532,6.023,148.941
C06912=1174.393,48.046,-48.404,-179.534,6.022,148.942
C06913=1174.398,47.796,-48.388,-179.537,6.021,148.942
C06914=1174.402,47.546,-48.373,-179.539,6.021,148.943
C06915=1174.408,47.297,-48.358,-179.543,6.019,148.943
C06916=1174.413,47.048,-48.341,-179.545,6.019,148.944
C06917=1174.418,46.798,-48.325,-179.547,6.018,148.944
C06918=1174.423,46.549,-48.310,-179.551,6.017,148.945
C06919=1174.428,46.300,-48.295,-179.553,6.016,148.946
C06920=1174.432,46.049,-48.279,-179.555,6.015,148.946
C06921=1174.438,45.800,-48.263,-179.557,6.014,148.947
C06922=1174.443,45.551,-48.248,-179.561,6.013,148.947
C06923=1174.448,45.302,-48.231,-179.563,6.012,148.948
C06924=1174.452,45.052,-48.216,-179.565,6.012,148.948
C06925=1174.458,44.803,-48.200,-179.568,6.011,148.949
C06926=1174.463,44.553,-48.185,-179.571,6.009,148.950
C06927=1174.467,44.303,-48.169,-179.574,6.009,148.950
C06928=1174.472,44.054,-48.154,-179.576,6.008,148.951
C06929=1174.478,43.805,-48.138,-179.579,6.007,148.951
C06930=1174.483,43.555,-48.123,-179.581,6.006,148.952
C06931=1174.487,43.305,-48.107,-179.584,6.005,148.952
C06932=1174.493,43.056,-48.092,-179.586,6.005,148.953
C06933=1174.498,42.807,-48.076,-179.589,6.003,148.954
C06934=1174.503,42.558,-48.061,-179.592,6.003,148.954
C06935=1174.507,42.307,-48.045,-179.594,6.002,148.955
C06936=1174.513,42.058,-48.030,-179.597,6.001,148.955
C06937=1174.518,41.809,-48.015,-179.600,6.000,148.956
C06938=1174.523,41.560,-47.999,-179.602,5.999,148.956
C06939=1174.528,41.309,-47.983,-179.605,5.999,148.957
C06940=1174.532,41.060,-47.968,-179.607,5.998,148.958
C06941=1174.538,40.811,-47.952,-179.610,5.997,148.958
C06942=1174.543,40.562,-47.937,-179.612,5.996,148.959
C06943=1174.548,40.312,-47.922,-179.615,5.995,148.959
C06944=1174.553,40.062,-47.906,-179.617,5.995,148.960
C06945=1174.558,39.813,-47.890,-179.620,5.994,148.961
C06946=1174.563,39.564,-47.875,-179.623,5.993,148.961
C06947=1174.568,39.314,-47.860,-179.625,5.992,148.962
C06948=1174.573,39.065,-47.845,-179.628,5.991,148.962
C06949=1174.578,38.815,-47.829,-179.630,5.991,148.963
C06950=1174.583,38.565,-47.814,-179.633,5.989,148.963
C06951=1174.588,38.316,-47.799,-179.636,5.989,148.964
C06952=1174.593,38.067,-47.783,-179.638,5.988,148.965
C06953=1174.598,37.818,-47.768,-179.640,5.987,148.965
C06954=1174.603,37.568,-47.753,-179.643,5.985,148.966
C06955=1174.608,37.319,-47.738,-179.646,5.985,148.966
C06956=1174.613,37.068,-47.723,-179.648,5.984,148.967
C06957=1174.618,36.819,-47.707,-179.651,5.984,148.967
C06958=1174.623,36.570,-47.692,-179.653,5.983,148.968
C06959=1174.628,36.321,-47.676,-179.656,5.981,148.969
C06960=1174.633,36.071,-47.662,-179.659,5.981,148.969
C06961=1174.639,35.821,-47.646,-179.661,5.980,148.970
C06962=1174.643,35.572,-47.631,-179.663,5.980,148.970
C06963=1174.648,35.322,-47.616,-179.667,5.978,148.971
C06964=1174.653,35.073,-47.601,-179.669,5.977,148.971
C06965=1174.658,34.823,-47.586,-179.671,5.977,148.972
C06966=1174.663,34.574,-47.571,-179.674,5.976,148.973
C06967=1174.669,34.325,-47.555,-179.676,5.976,148.973
C06968=1174.673,34.075,-47.541,-179.679,5.974,148.974
C06969=1174.679,33.826,-47.525,-179.682,5.973,148.974
C06970=1174.683,33.576,-47.510,-179.684,5.973,148.975
C06971=1174.688,33.327,-47.496,-179.687,5.972,148.976
C06972=1174.693,33.077,-47.480,-179.689,5.972,148.976
C06973=1174.698,32.828,-47.465,-179.692,5.970,148.977
C06974=1174.704,32.578,-47.450,-179.694,5.969,148.977
C06975=1174.708,32.328,-47.435,-179.697,5.969,148.978
C06976=1174.714,32.079,-47.420,-179.700,5.968,148.979
C06977=1174.719,31.829,-47.405,-179.702,5.968,148.979
C06978=1174.723,31.580,-47.390,-179.705,5.967,148.980
C06979=1174.729,31.330,-47.375,-179.707,5.965,148.980
C06980=1174.734,31.081,-47.360,-179.710,5.965,148.981
C06981=1174.739,30.832,-47.345,-179.713,5.964,148.982
C06982=1174.744,30.582,-47.331,-179.715,5.964,148.982
C06983=1174.749,30.333,-47.316,-179.717,5.963,148.983
C06984=1174.754,30.083,-47.301,-179.720,5.961,148.983
C06985=1174.759,29.834,-47.286,-179.723,5.961,148.984
C06986=1174.764,29.584,-47.270,-179.725,5.960,148.985
C06987=1174.769,29.335,-47.256,-179.728,5.960,148.985
C06988=1174.774,29.086,-47.241,-179.730,5.959,148.986
C06989=1174.780,28.836,-47.226,-179.732,5.958,148.986
C06990=1174.785,28.567,-47.210,-179.736,5.957,148.987
C06991=1174.790,28.298,-47.195,-179.738,5.957,148.987
C06992=1174.796,28.029,-47.178,-179.741,5.956,148.988
C06993=1174.801,27.760,-47.163,-179.744,5.955,148.989
C06994=1174.806,27.511,-47.147,-179.746,5.954,148.989
C06995=1174.811,27.261,-47.133,-179.749,5.953,148.990
C06996=1174.816,27.012,-47.118,-179.752,5.953,148.991
C06997=1174.821,26.762,-47.103,-179.754,5.952,148.991
C06998=1174.826,26.513,-47.088,-179.757,5.951,148.992
C06999=1174.831,26.263,-47.074,-179.759,5.950,148.992
C07000=1174.836,26.014,-47.059,-179.762,5.949,148.993
C07001=1174.841,25.764,-47.044,-179.764,5.949,148.994
C07002=1174.846,25.514,-47.029,-179.767,5.948,148.994
C07003=1174.851,25.265,-47.014,-179.769,5.948,148.995
C07004=1174.856,25.015,-47.000,-179.772,5.946,148.995
C07005=1174.861,24.766,-46.985,-179.775,5.945,148.996
C07006=1174.866,24.516,-46.970,-179.777,5.945,148.997
C07007=1174.871,24.267,-46.956,-179.779,5.944,148.997
C07008=1174.876,24.018,-46.941,-179.782,5.944,148.998
C07009=1174.881,23.768,-46.927,-179.785,5.943,148.998
C07010=1174.887,23.518,-46.912,-179.787,5.942,148.999
C07011=1174.891,23.269,-46.897,-179.790,5.941,148.999
C07012=1174.896,23.019,-46.883,-179.792,5.940,149.000
C07013=1174.902,22.770,-46.869,-179.795,5.940,149.001
C07014=1174.906,22.521,-46.854,-179.798,5.939,149.001
C07015=1174.912,22.271,-46.839,-179.800,5.938,149.002
C07016=1174.917,22.021,-46.825,-179.802,5.938,149.002
C07017=1174.922,21.771,-46.810,-179.805,5.937,149.003
C07018=1174.927,21.522,-46.795,-179.808,5.936,149.004
C07019=1174.932,21.273,-46.781,-179.811,5.935,149.004
C07020=1174.937,21.023,-46.767,-179.813,5.934,149.005
C07021=1174.942,20.773,-46.752,-179.815,5.934,149.005
C07022=1174.947,20.524,-46.737,-179.818,5.933,149.006
C07023=1174.952,20.275,-46.723,-179.820,5.933,149.007
C07024=1174.957,20.025,-46.709,-179.823,5.932,149.007
C07025=1174.962,19.775,-46.694,-179.825,5.932,149.008
C07026=1174.967,19.526,-46.679,-179.828,5.931,149.008
C07027=1174.972,19.277,-46.665,-179.831,5.929,149.009
C07028=1174.977,19.027,-46.651,-179.833,5.929,149.009
C07029=1174.983,18.777,-46.636,-179.836,5.928,149.010
C07030=1174.988,18.528,-46.622,-179.838,5.928,149.011
C07031=1174.993,18.278,-46.608,-179.840,5.927,149.011
C07032=1174.998,18.029,-46.593,-179.843,5.926,149.012
C07033=1175.003,17.779,-46.578,-179.846,5.926,149.013
C07034=1175.008,17.530,-46.564,-179.848,5.925,149.013
C07035=1175.013,17.280,-46.550,-179.851,5.924,149.014
C07036=1175.018,17.030,-46.536,-179.854,5.923,149.014
C07037=1175.023,16.781,-46.522,-179.856,5.922,149.015
C07038=1175.028,16.531,-46.507,-179.859,5.922,149.016
C07039=1175.033,16.282,-46.493,-179.861,5.921,149.016
C07040=1175.038,16.032,-46.479,-179.863,5.921,149.017
C07041=1175.043,15.782,-46.465,-179.866,5.920,149.017
C07042=1175.048,15.534,-46.450,-179.868,5.919,149.018
C07043=1175.053,15.284,-46.436,-179.871,5.919,149.019
C07044=1175.058,15.035,-46.421,-179.874,5.918,149.019
C07045=1175.063,14.785,-46.407,-179.876,5.917,149.020
C07046=1175.068,14.535,-46.393,-179.879,5.916,149.020
C07047=1175.074,14.286,-46.379,-179.881,5.915,149.021
C07048=1175.079,14.036,-46.365,-179.884,5.915,149.022
C07049=1175.084,13.787,-46.350,-179.886,5.914,149.022
C07050=1175.088,13.537,-46.336,-179.889,5.914,149.023
C07051=1175.094,13.288,-46.322,-179.891,5.913,149.023
C07052=1175.099,13.038,-46.308,-179.894,5.913,149.024
C07053=1175.104,12.789,-46.294,-179.896,5.912,149.024
C07054=1175.109,12.539,-46.279,-179.899,5.911,149.025
C07055=1175.114,12.289,-46.265,-179.901,5.911,149.026
C07056=1175.119,12.040,-46.251,-179.904,5.910,149.026
C07057=1175.125,11.790,-46.238,-179.906,5.909,149.027
C07058=1175.130,11.540,-46.223,-179.909,5.908,149.028
C07059=1175.135,11.291,-46.209,-179.912,5.907,149.028
C07060=1175.140,11.041,-46.195,-179.914,5.907,149.029
C07061=1175.145,10.792,-46.181,-179.916,5.906,149.029
C07062=1175.149,10.542,-46.167,-179.919,5.906,149.030
C07063=1175.155,10.293,-46.153,-179.922,5.905,149.031
C07064=1175.160,10.044,-46.139,-179.924,5.904,149.031
C07065=1175.165,9.794,-46.125,-179.927,5.904,149.032
C07066=1175.170,9.543,-46.111,-179.929,5.903,149.032
C07067=1175.176,9.294,-46.097,-179.931,5.902,149.033
C07068=1175.181,9.045,-46.083,-179.934,5.902,149.034
C07069=1175.185,8.795,-46.069,-179.937,5.901,149.034
C07070=1175.190,8.546,-46.055,-179.939,5.901,149.035
C07071=1175.195,8.297,-46.041,-179.941,5.900,149.035
C07072=1175.201,8.046,-46.028,-179.944,5.900,149.036
C07073=1175.206,7.797,-46.014,-179.947,5.898,149.037
C07074=1175.211,7.548,-45.999,-179.950,5.898,149.037
C07075=1175.216,7.298,-45.985,-179.952,5.897,149.038
C07076=1175.221,7.049,-45.972,-179.954,5.896,149.038
C07077=1175.226,6.799,-45.958,-179.957,5.896,149.039
C07078=1175.231,6.549,-45.944,-179.959,5.895,149.040
C07079=1175.237,6.300,-45.930,-179.962,5.894,149.040
C07080=1175.242,6.050,-45.916,-179.964,5.894,149.041
C07081=1175.246,5.800,-45.903,-179.967,5.893,149.041
C07082=1175.252,5.551,-45.889,-179.969,5.893,149.042
C07083=1175.257,5.302,-45.875,-179.972,5.892,149.043
C07084=1175.262,5.052,-45.860,-179.974,5.891,149.043
C07085=1175.267,4.803,-45.848,-179.977,5.891,149.044
C07086=1175.272,4.553,-45.833,-179.979,5.890,149.045
C07087=1175.277,4.303,-45.819,-179.982,5.890,149.045
C07088=1175.282,4.054,-45.806,-179.984,5.889,149.046
C07089=1175.287,3.804,-45.792,-179.987,5.889,149.046
C07090=1175.292,3.555,-45.778,-179.989,5.888,149.047
C07091=1175.297,3.305,-45.765,-179.992,5.887,149.048
C07092=1175.302,3.055,-45.751,-179.994,5.887,149.048
C07093=1175.307,2.806,-45.737,-179.997,5.886,149.049
C07094=1175.313,2.536,-45.723,-179.999,5.886,149.049
C07095=1175.318,2.267,-45.708,179.998,5.884,149.050
C07096=1175.324,1.998,-45.693,179.995,5.884,149.051
C07097=1175.330,1.729,-45.678,179.992,5.883,149.052
C07098=1175.334,1.479,-45.665,179.990,5.883,149.052
C07099=1175.340,1.230,-45.651,179.987,5.882,149.053
C07100=1175.345,0.980,-45.637,179.985,5.882,149.053
C07101=1175.349,0.730,-45.624,179.983,5.881,149.054
C07102=1175.355,0.481,-45.610,179.980,5.880,149.054
C07103=1175.360,0.231,-45.596,179.977,5.880,149.055
C07104=1175.365,-0.018,-45.583,179.975,5.879,149.056
C07105=1175.370,-0.268,-45.569,179.972,5.879,149.056
C07106=1175.376,-0.517,-45.556,179.970,5.878,149.057
C07107=1175.380,-0.767,-45.542,179.968,5.877,149.057
C07108=1175.386,-1.016,-45.529,179.965,5.877,149.058
C07109=1175.391,-1.266,-45.515,179.963,5.876,149.059
C07110=1175.395,-1.516,-45.502,179.960,5.875,149.059
C07111=1175.401,-1.765,-45.488,179.958,5.875,149.060
C07112=1175.406,-2.015,-45.475,179.955,5.874,149.060
C07113=1175.411,-2.264,-45.461,179.953,5.874,149.061
C07114=1175.416,-2.514,-45.448,179.950,5.873,149.062
C07115=1175.421,-2.764,-45.435,179.948,5.872,149.062
C07116=1175.426,-3.013,-45.421,179.945,5.872,149.063
C07117=1175.432,-3.263,-45.408,179.943,5.871,149.064
C07118=1175.436,-3.512,-45.394,179.940,5.871,149.064
C07119=1175.442,-3.762,-45.381,179.938,5.870,149.065
C07120=1175.447,-4.011,-45.367,179.935,5.870,149.066
C07121=1175.452,-4.261,-45.354,179.933,5.869,149.066
C07122=1175.457,-4.511,-45.341,179.930,5.868,149.067
C07123=1175.462,-4.760,-45.327,179.928,5.868,149.067
C07124=1175.467,-5.010,-45.314,179.925,5.867,149.068
C07125=1175.473,-5.260,-45.301,179.923,5.867,149.069
C07126=1175.477,-5.509,-45.287,179.920,5.866,149.069
C07127=1175.483,-5.759,-45.274,179.918,5.865,149.070
C07128=1175.487,-6.008,-45.260,179.915,5.865,149.070
C07129=1175.493,-6.258,-45.247,179.913,5.864,149.071
C07130=1175.498,-6.507,-45.234,179.910,5.864,149.072
C07131=1175.503,-6.757,-45.220,179.908,5.863,149.072
C07132=1175.508,-7.006,-45.207,179.905,5.863,149.073
C07133=1175.513,-7.256,-45.194,179.903,5.862,149.073
C07134=1175.519,-7.506,-45.181,179.900,5.861,149.074
C07135=1175.524,-7.756,-45.167,179.898,5.861,149.075
C07136=1175.529,-8.005,-45.154,179.895,5.860,149.075
C07137=1175.534,-8.255,-45.141,179.893,5.860,149.076
C07138=1175.539,-8.504,-45.127,179.890,5.859,149.077
C07139=1175.545,-8.753,-45.114,179.888,5.858,149.077
C07140=1175.549,-9.004,-45.101,179.885,5.858,149.078
C07141=1175.554,-9.253,-45.089,179.883,5.857,149.078
C07142=1175.560,-9.503,-45.075,179.881,5.857,149.079
C07143=1175.564,-9.752,-45.062,179.878,5.856,149.080
C07144=1175.570,-10.002,-45.048,179.876,5.856,149.080
C07145=1175.575,-10.252,-45.036,179.874,5.856,149.081
C07146=1175.580,-10.501,-45.023,179.871,5.855,149.081
C07147=1175.585,-10.751,-45.010,179.869,5.854,149.082
C07148=1175.590,-11.000,-44.996,179.866,5.854,149.083
C07149=1175.595,-11.250,-44.983,179.863,5.853,149.083
C07150=1175.600,-11.499,-44.970,179.861,5.853,149.084
C07151=1175.605,-11.749,-44.957,179.859,5.852,149.084
C07152=1175.611,-11.999,-44.944,179.856,5.852,149.085
C07153=1175.616,-12.248,-44.931,179.854,5.851,149.086
C07154=1175.621,-12.497,-44.918,179.851,5.850,149.086
C07155=1175.626,-12.747,-44.904,179.848,5.850,149.087
C07156=1175.631,-12.997,-44.892,179.846,5.849,149.087
C07157=1175.636,-13.246,-44.879,179.844,5.849,149.088
C07158=1175.641,-13.496,-44.866,179.841,5.848,149.089
C07159=1175.647,-13.746,-44.853,179.839,5.847,149.089
C07160=1175.651,-13.996,-44.840,179.836,5.847,149.090
C07161=1175.657,-14.245,-44.827,179.834,5.847,149.091
C07162=1175.662,-14.495,-44.814,179.831,5.846,149.091
C07163=1175.667,-14.745,-44.801,179.829,5.846,149.092
C07164=1175.672,-14.994,-44.788,179.827,5.846,149.093
C07165=1175.677,-15.243,-44.775,179.824,5.845,149.093
C07166=1175.682,-15.493,-44.762,179.822,5.844,149.094
C07167=1175.688,-15.743,-44.749,179.819,5.844,149.094
C07168=1175.693,-15.992,-44.736,179.817,5.843,149.095
C07169=1175.698,-16.241,-44.723,179.814,5.843,149.096
C07170=1175.702,-16.491,-44.710,179.812,5.842,149.096
C07171=1175.708,-16.741,-44.697,179.809,5.841,149.097
C07172=1175.713,-16.990,-44.685,179.807,5.841,149.097
C07173=1175.718,-17.240,-44.672,179.804,5.840,149.098
C07174=1175.723,-17.490,-44.659,179.802,5.840,149.099
C07175=1175.729,-17.740,-44.647,179.799,5.839,149.099
C07176=1175.734,-17.990,-44.634,179.797,5.839,149.100
C07177=1175.739,-18.239,-44.621,179.795,5.839,149.100
C07178=1175.744,-18.489,-44.608,179.792,5.838,149.101
C07179=1175.750,-18.738,-44.595,179.790,5.838,149.102
C07180=1175.754,-18.988,-44.582,179.788,5.837,149.102
C07181=1175.759,-19.238,-44.570,179.785,5.836,149.103
C07182=1175.765,-19.487,-44.557,179.782,5.836,149.104
C07183=1175.770,-19.736,-44.544,179.780,5.835,149.104
C07184=1175.775,-19.987,-44.531,179.777,5.835,149.105
C07185=1175.780,-20.236,-44.518,179.775,5.834,149.106
C07186=1175.785,-20.485,-44.506,179.773,5.833,149.106
C07187=1175.791,-20.735,-44.494,179.770,5.834,149.107
C07188=1175.795,-20.985,-44.481,179.768,5.833,149.107
C07189=1175.801,-21.235,-44.468,179.766,5.833,149.108
C07190=1175.806,-21.484,-44.455,179.763,5.832,149.109
C07191=1175.811,-21.733,-44.442,179.760,5.832,149.109
C07192=1175.816,-21.983,-44.430,179.758,5.831,149.110
C07193=1175.821,-22.233,-44.418,179.755,5.830,149.110
C07194=1175.826,-22.483,-44.405,179.753,5.830,149.111
C07195=1175.832,-22.732,-44.392,179.751,5.829,149.112
C07196=1175.837,-22.982,-44.379,179.748,5.829,149.112
C07197=1175.842,-23.232,-44.366,179.746,5.829,149.113
C07198=1175.848,-23.501,-44.354,179.744,5.828,149.113
C07199=1175.854,-23.771,-44.339,179.740,5.827,149.114
C07200=1175.859,-24.040,-44.326,179.738,5.827,149.115
C07201=1175.864,-24.310,-44.312,179.735,5.826,149.116
C07202=1175.870,-24.560,-44.300,179.733,5.826,149.116
C07203=1175.874,-24.810,-44.288,179.731,5.826,149.117
C07204=1175.879,-25.059,-44.275,179.728,5.825,149.117
C07205=1175.885,-25.310,-44.262,179.726,5.825,149.118
C07206=1175.891,-25.559,-44.250,179.723,5.824,149.119
C07207=1175.896,-25.808,-44.237,179.721,5.823,149.119
C07208=1175.901,-26.058,-44.225,179.718,5.823,149.120
C07209=1175.906,-26.308,-44.212,179.716,5.822,149.120
C07210=1175.911,-26.557,-44.200,179.713,5.822,149.121
C07211=1175.916,-26.807,-44.187,179.711,5.822,149.122
C07212=1175.921,-27.057,-44.175,179.709,5.821,149.122
C07213=1175.926,-27.306,-44.163,179.706,5.821,149.123
C07214=1175.932,-27.555,-44.150,179.704,5.820,149.124
C07215=1175.937,-27.805,-44.138,179.702,5.820,149.124
C07216=1175.941,-28.055,-44.125,179.699,5.819,149.125
C07217=1175.947,-28.305,-44.113,179.696,5.819,149.126
C07218=1175.952,-28.555,-44.101,179.695,5.819,149.126
C07219=1175.957,-28.804,-44.088,179.692,5.818,149.127
C07220=1175.963,-29.054,-44.076,179.689,5.818,149.127
C07221=1175.968,-29.303,-44.064,179.687,5.817,149.128
C07222=1175.973,-29.552,-44.051,179.684,5.817,149.129
C07223=1175.978,-29.802,-44.039,179.682,5.816,149.129
C07224=1175.983,-30.052,-44.026,179.680,5.815,149.130
C07225=1175.988,-30.302,-44.014,179.678,5.816,149.130
C07226=1175.993,-30.552,-44.002,179.675,5.815,149.131
C07227=1175.999,-30.802,-43.990,179.673,5.814,149.132
C07228=1176.004,-31.051,-43.977,179.670,5.814,149.132
C07229=1176.009,-31.301,-43.966,179.667,5.814,149.133
C07230=1176.014,-31.550,-43.953,179.665,5.813,149.134
C07231=1176.019,-31.799,-43.941,179.663,5.812,149.134
C07232=1176.024,-32.049,-43.929,179.660,5.813,149.135
C07233=1176.029,-32.298,-43.916,179.658,5.812,149.135
C07234=1176.035,-32.548,-43.904,179.656,5.811,149.136
C07235=1176.040,-32.798,-43.892,179.653,5.811,149.137
C07236=1176.045,-33.048,-43.880,179.651,5.810,149.137
C07237=1176.050,-33.298,-43.867,179.648,5.810,149.138
C07238=1176.055,-33.548,-43.855,179.646,5.809,149.138
C07239=1176.061,-33.798,-43.843,179.644,5.809,149.139
C07240=1176.065,-34.047,-43.831,179.641,5.809,149.140
C07241=1176.071,-34.296,-43.819,179.639,5.808,149.140
C07242=1176.076,-34.546,-43.807,179.636,5.808,149.141
C07243=1176.081,-34.796,-43.795,179.634,5.807,149.142
C07244=1176.086,-35.045,-43.782,179.631,5.806,149.142
C07245=1176.092,-35.295,-43.770,179.629,5.807,149.143
C07246=1176.097,-35.545,-43.758,179.627,5.806,149.144
C07247=1176.101,-35.794,-43.746,179.625,5.805,149.144
C07248=1176.107,-36.044,-43.735,179.622,5.805,149.145
C07249=1176.112,-36.293,-43.722,179.619,5.804,149.145
C07250=1176.117,-36.543,-43.710,179.617,5.804,149.146
C07251=1176.123,-36.793,-43.698,179.615,5.804,149.147
C07252=1176.128,-37.042,-43.686,179.612,5.804,149.147
C07253=1176.133,-37.292,-43.674,179.610,5.803,149.148
C07254=1176.138,-37.542,-43.662,179.607,5.802,149.148
C07255=1176.143,-37.791,-43.650,179.605,5.802,149.149
C07256=1176.149,-38.041,-43.638,179.603,5.802,149.150
C07257=1176.154,-38.291,-43.626,179.601,5.801,149.150
C07258=1176.159,-38.540,-43.614,179.598,5.801,149.151
C07259=1176.164,-38.790,-43.602,179.596,5.800,149.152
C07260=1176.169,-39.040,-43.590,179.593,5.800,149.152
C07261=1176.174,-39.289,-43.578,179.591,5.799,149.153
C07262=1176.180,-39.539,-43.566,179.589,5.799,149.153
C07263=1176.185,-39.789,-43.554,179.586,5.799,149.154
C07264=1176.190,-40.039,-43.543,179.584,5.798,149.155
C07265=1176.196,-40.287,-43.530,179.581,5.798,149.155
C07266=1176.201,-40.537,-43.518,179.579,5.797,149.156
C07267=1176.206,-40.787,-43.507,179.577,5.797,149.156
C07268=1176.211,-41.037,-43.495,179.574,5.797,149.157
C07269=1176.216,-41.286,-43.483,179.572,5.796,149.158
C07270=1176.221,-41.536,-43.471,179.570,5.796,149.158
C07271=1176.227,-41.786,-43.460,179.567,5.795,149.159
C07272=1176.232,-42.036,-43.448,179.565,5.795,149.160
C07273=1176.237,-42.285,-43.436,179.563,5.795,149.160
C07274=1176.242,-42.535,-43.424,179.560,5.794,149.161
C07275=1176.247,-42.785,-43.412,179.557,5.794,149.162
C07276=1176.253,-43.035,-43.400,179.555,5.793,149.162
C07277=1176.257,-43.284,-43.389,179.553,5.793,149.163
C07278=1176.263,-43.534,-43.377,179.550,5.793,149.163
C07279=1176.269,-43.783,-43.365,179.548,5.792,149.164
C07280=1176.273,-44.032,-43.353,179.546,5.792,149.165
C07281=1176.279,-44.282,-43.341,179.543,5.791,149.165
C07282=1176.284,-44.532,-43.329,179.541,5.791,149.166
C07283=1176.289,-44.782,-43.318,179.539,5.791,149.167
C07284=1176.294,-45.032,-43.306,179.536,5.790,149.167
C07285=1176.299,-45.281,-43.295,179.534,5.790,149.168
C07286=1176.304,-45.531,-43.283,179.532,5.790,149.168
C07287=1176.310,-45.781,-43.271,179.530,5.789,149.169
C07288=1176.315,-46.030,-43.260,179.527,5.789,149.170
C07289=1176.320,-46.280,-43.248,179.524,5.788,149.170
C07290=1176.326,-46.529,-43.236,179.522,5.787,149.171
C07291=1176.330,-46.779,-43.225,179.520,5.788,149.171
C07292=1176.336,-47.029,-43.213,179.517,5.787,149.172
C07293=1176.340,-47.279,-43.201,179.515,5.787,149.173
C07294=1176.346,-47.529,-43.189,179.512,5.786,149.173
C07295=1176.352,-47.778,-43.178,179.510,5.785,149.174
C07296=1176.357,-48.027,-43.167,179.508,5.786,149.175
C07297=1176.362,-48.277,-43.155,179.505,5.785,149.175
C07298=1176.367,-48.527,-43.144,179.503,5.785,149.176
C07299=1176.372,-48.777,-43.132,179.501,5.784,149.176
C07300=1176.377,-49.027,-43.120,179.499,5.784,149.177
C07301=1176.383,-49.276,-43.109,179.496,5.784,149.178
C07302=1176.388,-49.546,-43.096,179.494,5.783,149.178
C07303=1176.394,-49.817,-43.084,179.491,5.783,149.179
C07304=1176.400,-50.087,-43.071,179.488,5.782,149.180
C07305=1176.405,-50.358,-43.059,179.486,5.782,149.180
C07306=1176.410,-50.607,-43.047,179.484,5.781,149.181
C07307=1176.416,-50.857,-43.036,179.481,5.782,149.182
